FUNCTION_BLOCK "GCS7_M_Motors3W2HL"	// FB 48
TITLE = 3 Motors and 2 HL
//  
//COPYRIGHT:    (C) 1997  BUHLER AG, CH-9240 UZWIL, SWITZERLAND
//
//PRODUCT:      GCS7
//
//TITLE:        FB 48 Machine with 3 Motors and 2 HL 
//
//-------------------------------------------------------------------------
//
//IDENT:        AUTHOR:             DEPT:                       DATE:
//
//FB48.5.0      A. Egli             CT3                         17-Jul-2002
//              New Release with one block 
//              Condition Scraper.InLocal
//FB48.4.0      A. Egli             CT3                         24-Mai-2000
//              Element Scraper (FB11)
//              Mode Separator
//FB48.3.1      A. Egli             CT3                         30-Nov-1999
//              StFault = StCode 32
//FB48.3.0      A. Egli             CT3                         11-Oct-1999
//              Local data reduced 
//FB48.2B       K. Tischer          MU664                       06-Mrz-1999
//              CC FC2 not UC FC2
//FB48.2A       A. Egli             CT3                         04-Mai-1998
//              StFault = StCode 32
//FB48.1A       A.Egli              AEE61                       12-Nov-1997
//              1st Release in S7
//
//-------------------------------------------------------------------------
//
//PURPOSE:      MANUAL : see [LL.M3HxxMAN]
//
//RESTRICTIONS: S7
//              ACCU2: Pointer to dynamic datas of the machine
//              ACCU1: Pointer to parameter datas of the machine
//
//-------------------------------------------------------------------------
//
//
AUTHOR : EA
FAMILY : GCS7LL
NAME : Ma3M2HL
VERSION : 5.0
VAR
  Ma : UDT 20480;
  Motor1 : FB 12;	//Element
  Motor2 : FB 12;	//Element
  Motor3 : FB 12;	//Element
  HLLow : FB 14;	//Element
  HLInlet : FB 14;	//Element
  Scraper : FB 11;	//Element
END_VAR
VAR_TEMP
  tmpFaultStop : BOOL ;
  tmpFaultSum : BOOL ;
  tmpNext : BOOL ;
  tmpLocal : BOOL ;
  tmpEnable : BOOL ;
  tmpSeqStop : BOOL ;
  tmpLenDyn : INT ;
END_VAR
BEGIN
NETWORK
TITLE =
      L     10;
      T     #tmpLenDyn;
NETWORK
TITLE = PC Control
//=== Test Object number =====================
      L     "SYS_DirectCtrlDB".PC.ObjectNo;	//PCControl.ObjectNo
      L     #Ma.Par.ParObjectNo;	//Input ObjectNo
      <>I;
      JC    aEnd;
//=== Test OType      ========================
      L     2048;	//Input object type
      L     "SYS_DirectCtrlDB".PC.ObjectType;	//PCControl.ObjectType
      <>I;
      JC    aEnd;
//=== Test Handshake =========================
      A     "SYS_DirectCtrlDB".PC.Hsk.FExamine;	// Handshake.FExamine
      JC    aExa;
      A     "SYS_DirectCtrlDB".PC.Hsk.FDefineCmd;	// Handshake.FDefineCmd
      O     "SYS_DirectCtrlDB".PC.Hsk.FDefinePara;	// Handshake.FDefinePara
      JC    aCmd;
aIni: L     2;	// FcInit
      UC    "SYS_DirectCtrl";
      JU    aEnd;
// Write new commands from PC to Interface of group 
aCmd: A     "SYS_DirectCtrlDB".PC.Cmd1[0];	//Cmd1[0]=CmdOnM1
      S     #Ma.CmdOn;
      S     #Ma.InDisableM2;
      S     #Ma.InDisableM3;
      A     "SYS_DirectCtrlDB".PC.Cmd1[1];	//Cmd1[1]=CmdOnM2
      R     #Ma.InDisableM2;
      S     #Ma.CmdOn;
      A     "SYS_DirectCtrlDB".PC.Cmd2[1];	//Cmd2[1]=CmdOffM2
      S     #Ma.InDisableM2;
      A     "SYS_DirectCtrlDB".PC.Cmd1[2];	//Cmd1[2]=CmdOnM3
      R     #Ma.InDisableM3;
      S     #Ma.CmdOn;
      A     "SYS_DirectCtrlDB".PC.Cmd2[2];	//Cmd2[2]=CmdOffM3
      S     #Ma.InDisableM3;
      A     "SYS_DirectCtrlDB".PC.Cmd1[8];	//Cmd1[8]=CmdOff
      S     #Ma.CmdOff;
      A     "SYS_DirectCtrlDB".PC.Cmd1[9];	//Cmd1[9]=CmdOn
      S     #Ma.CmdOn;
      R     #Ma.InDisableM2;
      R     #Ma.InDisableM3;
      A     "SYS_DirectCtrlDB".PC.Cmd1[10];	//Cmd1[10]=CmdNext
      S     #Ma.CmdNext;
      A     "SYS_DirectCtrlDB".PC.Cmd1[11];	//Cmd1[11]=CmdFaultReset
      S     #Ma.CmdFaultReset;
      A     "SYS_DirectCtrlDB".PC.Cmd1[13];	//Cmd1[13]=CmdManualOn
      S     #Ma.InManual;
      A     "SYS_DirectCtrlDB".PC.Cmd2[13];	//Cmd1[13]=CmdManualOff
      R     #Ma.InManual;
      AN    "SYS_DirectCtrlDB".PC.Hsk.FDefinePara;	// Handshake.FDefinePara
      JC    aIni;
      JU    aIni;
aExa: TAR2;	// Address Dynamic data
      T     "SYS_DirectCtrlDB".GC.InDynAddr;	// -->PCControl.GC.InDynAddr
      L     #tmpLenDyn;	// Length Dynamic data
      T     "SYS_DirectCtrlDB".GC.InDynLen;	// -->PCControl.GC.InDynLen
      L     0;
      T     "SYS_DirectCtrlDB".GC.InParaAddr;	// -->PCControl.GC.InParaAddr
      T     "SYS_DirectCtrlDB".GC.InParaLen;	// -->PCControl.GC.InParaLen
      L     1;	// Code FcExamine
      UC    "SYS_DirectCtrl";
      L     10;	//Revision
      T     "SYS_DirectCtrlDB".GC.Revision;
aEnd: NOP   0;
NETWORK
TITLE = Interlocking
//===Global Group Orders===
      A     "GCS7_Gr_OutManualOn";	//Gr.OutManualOn
      S     #Ma.InManual;
      A     "GCS7_Gr_OutManualOff";	//Gr.OutManualOff
      R     #Ma.InManual;
      A     #Ma.InManual;
      S     "GCS7_Gr_InManual";	//Gr.InManual
      A     #Ma.CmdNext;
      AN    #Ma.InManual;
      O     #Ma.CmdOn;
      =     #tmpNext;
      A     #Ma.InManual;
      ON    #Ma.InLocal;
      A     #Ma.InEnable;
      AN    #Ma.CmdOff;
      =     #tmpEnable;
      A     #Ma.InSeqStop;
      AN    #Ma.InManual;
      =     #tmpSeqStop;
//--- Fault----
      A     #Motor1.StFault;
      O     #Motor2.StFault;
      O     #Motor3.StFault;
      O     #HLLow.StFault;
      O     #HLInlet.StFault;
      O     #Scraper.StFault;
      =     #tmpFaultSum;
//--- Next
      A(;
      A     #Motor2.StStartedFwd;
      ON    #Ma.Par.ParTypeSeparator;
      );
      A     #tmpNext;
      S     #Motor1.CmdNext;
      A     #Motor1.StStartedFwd;
      O     #Ma.Par.ParTypeSeparator;
      A     #tmpNext;
      S     #Motor2.CmdNext;
      S     #Motor3.CmdNext;
      A     #tmpNext;
      S     #Scraper.CmdNext;
//--- Interlocking Motors
//Motor1
      A     #tmpEnable;
      O     #Ma.Par.ParMotor1IsFan;
      =     #Motor1.InEnableFwd;
// 
      A     #tmpSeqStop;
      ON    #tmpEnable;
      A     #Motor2.StStopped;
      O;
      AN    #Ma.Par.ParMotor1IsFan;
      A     #tmpSeqStop;
      =     #Motor1.InSeqStop;
//Motor2
      AN    #HLLow.StFault;
      ON    #Ma.Par.ParWithHLLow;
      A(;
      A     #Motor1.StStartedFwd;
      O     #Ma.Par.ParTypeSeparator;
      );
      AN    #Ma.InDisableM2;
      A     #tmpEnable;
      =     #Motor2.InEnableFwd;
      A     #tmpSeqStop;
      =     #Motor2.InSeqStop;
//Motor3 
      A     #Motor2.InEnableFwd;
      A     #Motor2.StStartedFwd;
      O     #Ma.Par.ParTypeSeparator;
      A     #Motor1.StStartedFwd;
      AN    #Ma.InDisableM3;
      A     #tmpEnable;
      =     #Motor3.InEnableFwd;
      A     #tmpSeqStop;
      =     #Motor3.InSeqStop;
//Scraper
      A     #Motor2.StStartedFwd;
      A     #tmpEnable;
      =     #Scraper.InEnable;
      A     #tmpSeqStop;
      =     #Scraper.InSeqStop;
// 
//--- Local mode --
      A     #Ma.InLocal;
      AN    #Ma.InManual;
      =     #Motor1.InLocal;
      =     #Motor2.InLocal;
      =     #Motor3.InLocal;
      =     #HLLow.InLocal;
      =     #HLInlet.InLocal;
      =     #Scraper.InLocal;
//--- Fault Reset -------------
      A     #Ma.CmdFaultReset;
      S     #Motor1.CmdFaultReset;
      S     #Motor2.CmdFaultReset;
      S     #Motor3.CmdFaultReset;
      S     #HLLow.CmdFaultReset;
      S     #HLInlet.CmdFaultReset;
      S     #Scraper.CmdFaultReset;
// 
//--- Monitoring Level
      SET;
      S     #HLLow.InMonFalse;
      S     #HLInlet.InMonFalse;
NETWORK
TITLE = Call Motor1
      CALL  #Motor1;
NETWORK
TITLE = Call Motor2
      CALL  #Motor2;
NETWORK
TITLE = Call Motor3
      AN    #Ma.Par.ParWithMotor3;
      JC    el4;
      CALL  #Motor3;
NETWORK
TITLE = Call Digital Input: HLLow
el4:  AN    #Ma.Par.ParWithHLLow;
      JC    el5;
      CALL  #HLLow;
NETWORK
TITLE = Call Digital Input: HLInlet
el5:  AN    #Ma.Par.ParWithHLInlet;
      JC    el6;
      CALL  #HLInlet;
NETWORK
TITLE = Call Digital Output: Scraper
el6:  AN    #Ma.Par.ParWithScraper;
      JC    SPen;
      CALL  #Scraper;
SPen: NOP   0;
NETWORK
TITLE = Actual State
// StFault
      A     #tmpFaultSum;
      =     #Ma.StFault;
// StStopped
      A     #Motor3.StStopped;
      ON    #Ma.Par.ParWithMotor3;
      A     #Motor1.StStopped;
      A     #Motor2.StStopped;
      AN    #Ma.StFault;
      =     #Ma.StStopped;
// StStarted
      A     #Motor3.StStartedFwd;
      ON    #Ma.Par.ParWithMotor3;
      A     #Motor1.StStartedFwd;
      A     #Motor2.StStartedFwd;
      AN    #Ma.StFault;
      =     #Ma.StStarted;
// StStopping
      A     #Motor1.InSeqStop;
      O     #Motor2.InSeqStop;
      O     #Motor3.InSeqStop;
      AN    #Ma.StStarted;
      AN    #Ma.StStopped;
      AN    #Ma.StFault;
      =     #Ma.StStopping;
// StStarting
      AN    #Ma.StStopped;
      AN    #Ma.StStarted;
      AN    #Ma.StStopping;
      AN    #Ma.StFault;
      =     #Ma.StStarting;
NETWORK
TITLE = State Code
// State             StCode
// -------------------------
// StFault             32
// StStopped            1
// StStarting           2
// StStarted.Wait       3
// StStarted.Feeding    4
// StEmptying           5
// StEmptied            6
// StStopping           7
      A     #Ma.StStopped;
      L     1;	//Code=StStopped
      JC    Code;
      A     #Ma.StStarted;
      L     3;	//Code=StStarted
      JC    Code;
      A     #Ma.StStarting;
      L     2;	//Code=StStarting
      JC    Code;
      A     #Ma.StStopping;
      L     7;	//Code=StStopping 
      JC    Code;
      L     32;	//3.1: Code=StFault 
Code: L     #Ma.StCode;	// Old state code
      TAK;
      T     #Ma.StCode;	// Save state code
      <>I;
      L     3;
      CC    "SYS_CBitCtrl";	//Set change bit
NETWORK
TITLE = Global End
      CLR;	//---Clear all commands
      =     #Ma.CmdOn;
      =     #Ma.CmdOff;
      =     #Ma.CmdNext;
      =     #Ma.CmdFaultReset;
END_FUNCTION_BLOCK

FUNCTION_BLOCK "GCS7_M_MDDX"	// FB 49
TITLE = MDDx Newtronic Roll Stand
//  
//COPYRIGHT:    (C) 1999  BUHLER AG, CH-9240 UZWIL, SWITZERLAND
//
//PRODUCT:      GCS7
//
//TITLE:        FB 49 Machine MDDx Newtronic Roll Stand
//              (GCPROVB Revision 11)
//-------------------------------------------------------------------------
//
//IDENT:        AUTHOR:             DEPT:                       DATE:
//
//FB49.5.3      A. Egli             CT3                         15-Aug-2007
//              MDDX.OutComFault stops motors
//FB49.5.2      A. Egli             CT3                         15-Feb-2007
//              Stop Motors when alarm 14 or 15
//FB49.5.1      Ph. Enger           MU664                       21-Sep-2004
//              Interlocking with BackupHL corrected
//FB49.5.0      Ph. Enger           MU664                       16-Sep-2004
//              New configuration ParB1
//FB49.4.0      A. Egli             CT3                         28-Jul-2004
//              New Version of FB35
//FB49.3.1      A. Egli             CT3                         05-Mai-2004
//              CmdOff in manual mode
//FB49.3.0      A. Egli             CT3                         17-Jul-2002
//              New Release with one block 
//FB49.2.2      A. Egli             CT3                         18-Mai-2000
//              CBIT: UC changed with CC 
//FB49.2.1      S. Kalberer         CT3                         29-Nov-1999
//              HLInlet: InOverwriteHL function to InMonFalse not InLocal
//FB49.2.0      A. Egli             CT3                         11-Oct-1999
//              Local data reduced 
//FB49.1A       S. Kalberer         CT3                         30-Jul-1999
//              1st Release in S7
//
//-------------------------------------------------------------------------
//
//PURPOSE:      MANUAL : see [LL.ROXENMAN]
//
//RESTRICTIONS: S7
//              ACCU2: Pointer to dynamic datas of the machine
//              ACCU1: Pointer to parameter datas of the machine
//
//-------------------------------------------------------------------------
//
//
AUTHOR : EA
FAMILY : GCS7LL
NAME : MDDxNtro
VERSION : 5.3
VAR
  Ma : UDT 20490;
  RollsUp : FB 12;	//Element
  RollsLow : FB 12;	//Element
  HLInlet : FB 14;	//Element
  HLBackUp : FB 14;	//Element
  HLOutlet : FB 14;	//Element
  CollectAlarm : FB 14;	//Element
  MddLC : FB 35;	//Element
  FU_Feedroll : FB 14;	//Element FU Feedroll [3.0]
END_VAR
VAR_TEMP
  tmpFaultSum : BOOL ;
  tmpWarning : BOOL ;
  tmpStarted : BOOL ;
  tmpNext : BOOL ;
  tmpLocal : BOOL ;
  tmpEnable : BOOL ;
  tmpSeqStop : BOOL ;
  tmpLenDyn : INT ;
END_VAR
BEGIN
NETWORK
TITLE =
      L     10;
      T     #tmpLenDyn;
NETWORK
TITLE = PC Control
//=== Test Object number =====================
      L     "SYS_DirectCtrlDB".PC.ObjectNo;	//PCControl.ObjectNo
      L     #Ma.Par.ParObjectNo;	//Input ObjectNo
      <>I;
      JC    aEnd;
//=== Test OType      ========================
      L     2049;	//Input object type
      L     "SYS_DirectCtrlDB".PC.ObjectType;	//PCControl.ObjectType
      <>I;
      JC    aEnd;
//=== Test Handshake =========================
      A     "SYS_DirectCtrlDB".PC.Hsk.FExamine;	// Handshake.FExamine
      JC    aExa;
      A     "SYS_DirectCtrlDB".PC.Hsk.FDefineCmd;	// Handshake.FDefineCmd
      O     "SYS_DirectCtrlDB".PC.Hsk.FDefinePara;	// Handshake.FDefinePara
      JC    aCmd;
aIni: L     2;	// FcInit
      UC    "SYS_DirectCtrl";
      JU    aEnd;
// Write new commands from PC to Interface of group 
aCmd: A     "SYS_DirectCtrlDB".PC.Cmd1[1];	//Cmd1[1]=CmdEnableEngageOn
      S     #Ma.InEnableEngage;
      A     "SYS_DirectCtrlDB".PC.Cmd2[1];	//Cmd2[1]=CmdEnableEngageOff
      R     #Ma.InEnableEngage;
      A     "SYS_DirectCtrlDB".PC.Cmd1[2];	//Cmd1[2]=CmdResDischargeOn
      S     #Ma.InRestdischarge;
      A     "SYS_DirectCtrlDB".PC.Cmd2[2];	//Cmd2[2]=CmdRestDischargeOff
      R     #Ma.InRestdischarge;
      A     "SYS_DirectCtrlDB".PC.Cmd1[3];	//Cmd1[3]=CmdOverwriteHLOn
      S     #Ma.InOverrideHL;
      A     "SYS_DirectCtrlDB".PC.Cmd2[3];	//Cmd2[3]=CmdOverwriteHLOff
      R     #Ma.InOverrideHL;
      A     "SYS_DirectCtrlDB".PC.Cmd1[8];	//Cmd1[8]=CmdOff
      S     #Ma.CmdOff;
      A     "SYS_DirectCtrlDB".PC.Cmd1[9];	//Cmd1[9]=CmdOn
      S     #Ma.CmdOn;
      A     "SYS_DirectCtrlDB".PC.Cmd1[10];	//Cmd1[10]=CmdNext
      S     #Ma.CmdNext;
      A     "SYS_DirectCtrlDB".PC.Cmd1[11];	//Cmd1[11]=CmdFaultReset
      S     #Ma.CmdFaultReset;
      A     "SYS_DirectCtrlDB".PC.Cmd1[13];	//Cmd1[13]=CmdManualOn
      S     #Ma.InManual;
      A     "SYS_DirectCtrlDB".PC.Cmd2[13];	//Cmd1[13]=CmdManualOff
      R     #Ma.InManual;
      AN    "SYS_DirectCtrlDB".PC.Hsk.FDefinePara;	// Handshake.FDefinePara
      JC    aIni;
      JU    aIni;
aExa: TAR2;	// Address Dynamic data
      T     "SYS_DirectCtrlDB".GC.InDynAddr;	// -->PCControl.GC.InDynAddr
      L     #tmpLenDyn;	// Length Dynamic data
      T     "SYS_DirectCtrlDB".GC.InDynLen;	// -->PCControl.GC.InDynLen
      L     0;
      T     "SYS_DirectCtrlDB".GC.InParaAddr;	// -->PCControl.GC.InParaAddr
      T     "SYS_DirectCtrlDB".GC.InParaLen;	// -->PCControl.GC.InParaLen
      L     1;	// Code FcExamine
      UC    "SYS_DirectCtrl";
      L     12;	//Revision
      T     "SYS_DirectCtrlDB".GC.Revision;
aEnd: NOP   0;
NETWORK
TITLE = Interlocking
//===Global Group Orders===
      A     "GCS7_Gr_OutManualOn";	//Gr.OutManualOn
      S     #Ma.InManual;
      A     "GCS7_Gr_OutManualOff";	//Gr.OutManualOff
      R     #Ma.InManual;
      A     #Ma.InManual;
      S     "GCS7_Gr_InManual";	//Gr.InManual
//--- temporary Next ---
      AN    #Ma.StStarting;
      ON    #Ma.InManual;
      O     #Ma.CmdOff;	//[3.1]
      R     #Ma.OutStartMan;
      O     #Ma.CmdOn;
      S     #Ma.OutStartMan;
      A     #Ma.CmdNext;
      AN    #Ma.InManual;
      O     #Ma.OutStartMan;
      =     #tmpNext;
//--- temporary Enable ---
      A(;
      A     #Ma.InEnable;
      AN    #Ma.InLocal;
      AN    #Ma.InManual;
      O;
      A     #Ma.InEnable;
      A     #Ma.InManual;
      AN    #Ma.Par.ParManual;
      O;
      A     #Ma.Par.ParManual;
      A     #Ma.InManual;
      );
      AN    #Ma.CmdOff;
      AN    #MddLC.Par.OutLCAlarm.GrindRollsStandstill;	//[5.2]
      AN    #MddLC.Par.OutLCAlarm.GrindRollsLowStandstill;	//[5.2]
      AN    #MddLC.OutComFault;	//[5.3]
      =     #tmpEnable;
//--- temporary SeqStop ---
      A     #Ma.InSeqStop;
      AN    #Ma.InManual;
      =     #tmpSeqStop;
//--- Fault----
      A     #RollsUp.StFault;
      O     #RollsLow.StFault;
      =     #tmpWarning;
      A     #tmpWarning;
      AN    #Ma.Par.ParWarning;
      O     #HLBackUp.StFault;
      O     #HLInlet.StFault;
      O     #HLOutlet.StFault;
      O     #CollectAlarm.StFault;
      O     #MddLC.StFault;
      O     #FU_Feedroll.StFault;	//[3.0]
      =     #tmpFaultSum;
//--- Next
      A     #HLBackUp.StFalse;	//[5.0]
      ON    #Ma.Par.ParWithHLBackUp;	//[5.1]
      A     #tmpNext;
      S     #RollsLow.CmdNext;
      S     #RollsUp.CmdNext;
//--- Interlocking Motors
//RollsLow
      A     #tmpEnable;
      AN    #tmpSeqStop;	//[5.0]
      =     #RollsLow.InEnableFwd;
// 
      A     #HLBackUp.StFault;	//[5.0]
      A     #HLBackUp.InpTrue;	//[5.0]
      =     #RollsLow.InSeqStop;
//RollsUp
      A     #RollsLow.StStartedFwd;
      ON    #Ma.Par.ParWithRollsLow;
      A     #tmpEnable;
      AN    #tmpSeqStop;	//[5.0]
      =     #RollsUp.InEnableFwd;
      A     #HLBackUp.StFault;	//[5.0]
      A     #HLBackUp.InpTrue;	//[5.0]
      =     #RollsUp.InSeqStop;
//--- Local mode --
      A     #Ma.InLocal;
      AN    #Ma.InManual;
      =     #RollsLow.InLocal;
      =     #RollsUp.InLocal;
      =     #HLBackUp.InLocal;
      =     #HLOutlet.InLocal;
      =     #CollectAlarm.InLocal;
      =     #MddLC.InLocal;
      =     #FU_Feedroll.InLocal;	//[3.0]
//        U     #Ma.InLocal;      // 2.1
//        UN    #Ma.InManual;     // 2.1
//        O     #Ma.InOverwriteHL; // 2.1 
      =     #HLInlet.InLocal;
//--- Fault Reset -------------
      A     #Ma.CmdFaultReset;
      S     #RollsLow.CmdFaultReset;
      S     #RollsUp.CmdFaultReset;
      S     #HLInlet.CmdFaultReset;
      S     #HLBackUp.CmdFaultReset;
      S     #HLOutlet.CmdFaultReset;
      S     #CollectAlarm.CmdFaultReset;
      S     #MddLC.CmdFaultReset;
      S     #FU_Feedroll.CmdFaultReset;	//[3.0]
//--- Monitoring 
      AN    #Ma.InOverrideHL;	// 2.1
      O     #Ma.Par.ParB1;	//[5.0]
      =     #HLInlet.InMonFalse;	// 2.1
      AN    #Ma.Par.ParB1;	//[5.0]
      AN    #Ma.InOverrideHL;	//[5.0]
      =     #HLInlet.InPreAlarmFalse;	//[5.0]
// 
      A     #HLInlet.OutFlagPos;	//[5.0] 
      AN    #HLInlet.OutTimeoutTime;	//[5.0] 
      A     #Ma.Par.ParB1;	//[5.0]
      S     #HLInlet.CmdRunTimeoutTime;	//[5.0]
// 
      SET;
      S     #HLBackUp.InMonFalse;
      S     #HLOutlet.InMonFalse;
      S     #CollectAlarm.InMonTrue;
//Startup done
      A     #RollsUp.StStartedFwd;
      O     #RollsUp.StFault;
      A(;
      A     #RollsLow.StStartedFwd;
      O     #RollsLow.StFault;
      ON    #Ma.Par.ParWithRollsLow;
      );
      =     #Ma.OutStartupDone;
      A     #RollsLow.StStartedFwd;
      ON    #Ma.Par.ParWithRollsLow;
      A     #RollsUp.StStartedFwd;
      =     #tmpStarted;
//--- Serial Communication Handling
// EnableEngage
      A     #Ma.InEnable;
      AN    #Ma.InLocal;
      AN    #Ma.InManual;
      O     #Ma.InEnableEngage;
      =     #MddLC.InEnableEngage;
//  RestDischarge
      A     #Ma.InRestdischarge;
      =     #MddLC.InRestdischarge;
NETWORK
TITLE = Call RollsUp
      CALL  #RollsUp;
NETWORK
TITLE = Call RollsLow
      AN    #Ma.Par.ParWithRollsLow;
      JC    el3;
      CALL  #RollsLow;
NETWORK
TITLE = Call Digital Input: HLInlet
el3:  AN    #Ma.Par.ParWithHLInlet;
      JC    el4;
      CALL  #HLInlet;
NETWORK
TITLE = Call Digital Input: HLBackUp
el4:  AN    #Ma.Par.ParWithHLBackUp;
      JC    el5;
      CALL  #HLBackUp;
NETWORK
TITLE = Call Digital Input: HLOutlet
el5:  AN    #Ma.Par.ParWithHLOutlet;
      JC    el6;
      CALL  #HLOutlet;
NETWORK
TITLE = Call Digital Input: CollectAlarm
el6:  AN    #Ma.Par.ParWithCollectAlarm;
      JC    el7;
      CALL  #CollectAlarm;
NETWORK
TITLE = Call MDDx Serial Communication: MddLC
el7:  AN    #Ma.Par.ParWithMddLC;
      JC    el8;
      CALL  #MddLC;
NETWORK
TITLE = Call MDDx Serial Communication: MddLC
el8:  AN    #Ma.Par.ParWithFU_FeedRoll;	//[3.0]
      JC    StJ0;
      CALL  #FU_Feedroll;
NETWORK
TITLE = Actual State
// StFault
StJ0: A     #tmpFaultSum;
      =     #Ma.StFault;
// StWarning
      A     #tmpWarning;
      A     #Ma.Par.ParWarning;
      AN    #Ma.StFault;
      O     #MddLC.StWarning;
      =     #Ma.StWarning;
// StStopped
      A     #RollsLow.StStopped;
      ON    #Ma.Par.ParWithRollsLow;
      A     #RollsUp.StStopped;
      AN    #Ma.StFault;
      =     #Ma.StStopped;
// StStarted
      A     #tmpStarted;
      AN    #Ma.StFault;
      AN    #Ma.StStopped;
      =     #Ma.StStarted;
// StStopping
      A     #RollsUp.InSeqStop;
      O     #RollsLow.InSeqStop;
      AN    #Ma.StStarted;
      AN    #Ma.StStopped;
      AN    #Ma.StFault;
      AN    #Ma.StWarning;
      =     #Ma.StStopping;
// StStarting
      AN    #Ma.StStopped;
      AN    #Ma.StStarted;
      AN    #Ma.StStopping;
      AN    #Ma.StFault;
      AN    #Ma.StWarning;
      =     #Ma.StStarting;
NETWORK
TITLE = State Code
// State     StCode
// ----------------------
// StFault32
// StStopped    1
// StStarting   2
// StStarted   3
// StStopping  7
// StWarning8
      A     #Ma.StStopped;
      L     1;	//Code=StStopped
      JC    Code;
      A     #Ma.StStarted;
      L     3;	//Code=StStarted
      JC    Code;
      A     #Ma.StWarning;
      L     8;	//Code=StWarning 
      JC    Code;
      A     #Ma.StStarting;
      L     2;	//Code=StStarting
      JC    Code;
      A     #Ma.StStopping;
      L     7;	//Code=StStopping 
      JC    Code;
      L     32;	//Code=StFault 
Code: L     #Ma.StCode;	// Old state code
      TAK;
      T     #Ma.StCode;	// Save state code
      <>I;
      L     3;
      CC    "SYS_CBitCtrl";	//Set change bit [REL 2.2]
NETWORK
TITLE = Global End
      CLR;	//---Clear all commands
      =     #Ma.CmdOn;
      =     #Ma.CmdOff;
      =     #Ma.CmdNext;
      =     #Ma.CmdFaultReset;
END_FUNCTION_BLOCK

FUNCTION_BLOCK "GCS7_M_Motor6Mon"	// FB 50
TITLE = Motor with 6 digital input
//  
//COPYRIGHT:    (C) 1997  BUHLER AG, CH-9240 UZWIL,  SWITZERLAND
//
//PRODUCT:      GCS7
//
//TITLE:        FB 50 MACHINE-CONTROL:Motor with 6 Digital input 
//              GCPROVB Revision >=12
// 
//-------------------------------------------------------------------------
//
//IDENT:        AUTHOR:             DEPT:                       DATE:
//FB50.8.6      A.Egli              BASE                        10-Apr-2008
//              - Init if download DB
//              - Condition MonX.InLocal 
//FB50.8.5      Ph. Engler          GP92                        23-Aug-2007
//              Machine status: StStarting how long the monitoring elements
//FB50.8.5      Ph. Engler          GP92                        23-Aug-2007
//              Machine status: StStarting how long the monitoring elements
//                              aren't in the correct status
//FB50.8.4      A.Egli              CT3                         20-Feb-2006
//              EBM-Test procedure: - Include als the EBMInput to the test
//                                  - Manual and local mode also integrated 
//              (Tested Ph.Engler, GP92,24-Aug-2005 )
//FB50.8.3      A.Egli              CT3                         09-Mar-2005
//              Send CmdFaultReset only with positve edge to elements  
//FB50.8.2      A.Egli              CT3                         20-Sep-2004 
//              Delay time before and between 2 single tests of EBM  
//FB50.8.1      A.Egli              CT3                         20-Jul-2004
//              tmpLenDyn is 12 and not 10
//FB50.8.0      A.Egli              CT3                         25-Mai-2004
//              ParMon4IsSM
//FB50.7.6      A.Egli              CT3                         15-Apr-2004
//              Test with Hardware 
//FB50.7.5      A.Egli              CT3                         18-Mar-2004
//              InpControlEBM 
//FB50.7.4      K. Tischer          CT3                         13-Feb-2004
//              interlocking without Mon1 
//FB50.7.3      K. Tischer          CT3                         30-Jan-2004
//              Correct monitoring Mon4 
//FB50.7.2      K. Tischer          CT3                         14-Jan-2004
//              Revision=11 
//FB50.7.1      K. Tischer          CT3                         02-Dec-2003
//              new 6 DI and supported EBM3003 
//FB50.7.0      K. Tischer          CT3                         01-Dec-2003
//              new 6 DI and supported EBM3003 
//FB50.6.2      A. Egli             CT3                         22-Sep-2003
//              Interlocking Mon4.StFalse when Mon4 is HL
//FB50.6.1      A. Egli             CT3                         16-Mai-2003
//              Interlocking if Mon1 is HL
//              Send CmdOff to Motor
//FB50.6.0      A. Egli             CT3                         17-Jun-2002
//              New Release with one block 
//              Interlocking if Mon1 is HL
//FB50.5.0      A. Egli             CT3                          1-Feb-2002
//              -HLInlet renamed as Mon4
//              -ParMon4StopByFault,ParMon4IsLS
//FB50.4.0      A. Egli             CT3                         15-Jan-2002
//              HLIntet as Warning Element
//FB50.3.1      A. Egli             CT3                         23-Oct-2001
//              Manual Mode: no interlocking with InSeqStop
//FB50.3.0      A. Egli             CT3                         11-Oct-1999
//              Local data reduced 
//FB50.2C       A. Egli             CT3                         03-Juni-1999
//              Manual Mode
//FB50.2B       K. Tischer          MU664                       06-Mrz-1999
//              CC FC2 not UC FC2
//FB50.2A       A. Egli             CT3                         04-Mai-1998
//              StFault = StCode 32
//FB50.1A       A.Egli              AEE61                       5-Jul-1997
//              1st Release in S7
//
//-------------------------------------------------------------------------
//
//PURPOSE:      MANUAL : see [LL.M4IxxMAN]
//
//RESTRICTIONS: S7
//
//              GCPROVB Revision >=5
//-------------------------------------------------------------------------
//
AUTHOR : EA
FAMILY : GCS7LL
NAME : M_6DI
VERSION : 8.6
VAR
  Ma : UDT 20500;
  Mon1 : FB 14;	//Element Mon 1 optional
  Mon2 : FB 14;	//Element Mon 2
  Mon3 : FB 14;	//Element Mon 3 optional
  Mon4 : FB 14;	//Element Mon 4 optional
  Mon5 : FB 14;	//Element Mon 5 optional [7.0]
  Mon6 : FB 14;	//Element Mon 6 optional [7.0]
  Motor : FB 12;	//Element Motor
END_VAR
VAR_TEMP
  tmpFaultStop : BOOL ;
  tmpFaultSum : BOOL ;
  tmpEnable : BOOL ;
  tmpLocal : BOOL ;
  tmpLenDyn : INT ;
  tmpOK : BOOL ;
  tmpTestTime : INT ;
  tmpMonElOk : BOOL ;
END_VAR
BEGIN
NETWORK
TITLE =
      L     12;
      T     #tmpLenDyn;	//[8.1]
NETWORK
TITLE = PC Control
//=== Test Object number =====================
      L     "SYS_DirectCtrlDB".PC.ObjectNo;	//PCControl.ObjectNo
      L     #Ma.Par.ParObjectNo;	//Input ObjectNo
      <>I;
      JC    aEnd;
//=== Test OType      ========================
      L     2050;	//Input object type
      L     "SYS_DirectCtrlDB".PC.ObjectType;	//PCControl.ObjectType
      <>I;
      JC    aEnd;
//=== Test Handshake =========================
      A     "SYS_DirectCtrlDB".PC.Hsk.FExamine;	// Handshake.FExamine
      JC    aExa;
      A     "SYS_DirectCtrlDB".PC.Hsk.FDefineCmd;	// Handshake.FDefineCmd
      O     "SYS_DirectCtrlDB".PC.Hsk.FDefinePara;	// Handshake.FDefinePara
      JC    aCmd;
aIni: L     2;	// FcInit
      UC    "SYS_DirectCtrl";
      JU    aEnd;
// Write new commands from PC to Interface of group 
aCmd: A     "SYS_DirectCtrlDB".PC.Cmd1[8];	//Cmd1[8]=CmdOff
      S     #Ma.CmdOff;
      A     "SYS_DirectCtrlDB".PC.Cmd1[9];	//Cmd1[9]=CmdOn
      S     #Ma.CmdOn;
      A     "SYS_DirectCtrlDB".PC.Cmd1[10];	//Cmd1[10]=CmdNext
      S     #Ma.CmdNext;
      A     "SYS_DirectCtrlDB".PC.Cmd1[11];	//Cmd1[11]=CmdFaultReset
      S     #Ma.CmdFaultReset;
      A     "SYS_DirectCtrlDB".PC.Cmd1[13];	//Cmd1[13]=CmdManualOn
      S     #Ma.InManual;
      A     "SYS_DirectCtrlDB".PC.Cmd1[6];	//Cmd1[6]=CmdManSlowOn
      S     #Motor.InOutManSlow;
      A     "SYS_DirectCtrlDB".PC.Cmd1[7];	//Cmd1[7]=CmdManRevOn
      S     #Motor.InOutManRev;
      A     "SYS_DirectCtrlDB".PC.Cmd2[13];	//Cmd2[13]=CmdManualOff
      R     #Ma.InManual;
      A     "SYS_DirectCtrlDB".PC.Cmd2[6];	//Cmd2[6]=CmdManSlowOff
      R     #Motor.InOutManSlow;
      A     "SYS_DirectCtrlDB".PC.Cmd2[7];	//Cmd2[7]=CmdManRevOff
      R     #Motor.InOutManRev;
      JU    aIni;
aExa: TAR2;	// Address Dynamic datas
      T     "SYS_DirectCtrlDB".GC.InDynAddr;	// -->PCControl.GC.InDynAddr
      L     #tmpLenDyn;	// Length Dynamic data
      T     "SYS_DirectCtrlDB".GC.InDynLen;	// -->PCControl.GC.InDynLen
      L     0;
      T     "SYS_DirectCtrlDB".GC.InParaAddr;	// -->PCControl.GC.InParaAddr
      T     "SYS_DirectCtrlDB".GC.InParaLen;	// -->PCControl.GC.InParaLen
      L     1;	// Code FcExamine
      UC    "SYS_DirectCtrl";
      L     12;	//Revision
      T     "SYS_DirectCtrlDB".GC.Revision;
aEnd: NOP   0;
NETWORK
TITLE = function test [7.0]
      L     720;	//[8.2] 
      T     #tmpTestTime;	//[8.2] 
      AN    #Ma.Par.ParEBM;
      JC    FCT0;
      A     #Ma.InLocal;
      AN    #Ma.InManual;
      =     #tmpLocal;
      L     0;
      L     #Ma.OutTestTime;
      >=I;
      O     #Ma.CmdTestEBM;
      R     #Ma.InfBMTopOk;
      R     #Ma.InfBMBottomOk;
      R     #Ma.InfSMOk;
      R     #Ma.CmdTestEBM;
      L     #tmpTestTime;	//s = 12min 
      JC    FCT;
      AN    #Motor.StStartedFwd;	//[8.2] 
      AN    #Motor.StStartedRev;	//[8.2] 
      AN    #Ma.InfSMOk;	//[8.2] 
      L     #tmpTestTime;	//[8.2] 
      JC    FCT;	//[8.2] 
      L     #Ma.OutTestTime;
      AN    "GCS7_Gr_OutTick1s";	// Gr.OutTick1s
      JC    FCT;
      +     -1;
FCT:  T     #Ma.OutTestTime;
// function test SM
      L     #tmpTestTime;	//[8.2] 
      L     #Ma.OutTestTime;	//[8.2] 
      -I;	//[8.2] 
      L     35;	//[8.2] 
      >=I;	//[8.2] 
      A     #Ma.InpControlEBM;	//[7.5]
      AN    #Ma.OutpFaultReset;	//[7.5]
      AN    #Ma.StFault;	//[7.5]
      O     #Ma.OutpFcttst_SM;	//[7.5]
      AN    #Ma.InfSMOk;
      AN    #Mon1.InLocal;
      AN    #Ma.StStopped;	//[8.2]
      =     #Ma.OutpFcttst_SM;
// function test ok SM
      A     #Ma.OutpFcttst_SM;
      A(;
      ON    #Mon6.InpTrue;
      ON    #Ma.Par.ParWithMon6;
      );
      AN    #Ma.InpControlEBM;	//[7.5]
      =     #tmpOK;	//[7.5]
      A     #tmpOK;	//[7.5]
      AN    #Ma.InfSMOk;	//[7.5]
      S     #Ma.InfSMOk;
      S     #Ma.OutFaultResetFcttst;	//[7.5]
      JCN   BTJ1;	//[8.2] 
      L     #tmpTestTime;	//[8.2] s = 12min 
      T     #Ma.OutTestTime;	//[8.2] 
BTJ1: NOP   0;	//[8.2] 
// function test BM top
      L     #tmpTestTime;	//[8.2] s = 12min 
      L     #Ma.OutTestTime;	//[8.2] 
      -I;	//[8.2] 
      L     5;	//[8.2] 
      >=I;	//[8.2] 
      AN    #Ma.OutpFaultReset;	//[7.5]
      A     #Ma.InpControlEBM;	//[7.5]
      AN    #Ma.StFault;	//[7.5]
      O     #Ma.OutpFcttst_BM_Top;	//[7.5]
      AN    #Ma.InfBMTopOk;
      A     #Ma.InfSMOk;	//[7.6]
      AN    #Mon1.InLocal;
      =     #Ma.OutpFcttst_BM_Top;
// function test ok
      A     #Ma.OutpFcttst_BM_Top;
      AN    #Mon2.InpTrue;
      AN    #Ma.InpControlEBM;	//[7.5]
      =     #tmpOK;	//[7.5]
      A     #tmpOK;	//[7.5]
      AN    #Ma.InfBMTopOk;	//[7.5]
      S     #Ma.InfBMTopOk;
      S     #Ma.OutFaultResetFcttst;	//[7.5]
      JCN   BTJ2;	//[8.2] 
      L     #tmpTestTime;	//[8.2] s = 12min 
      T     #Ma.OutTestTime;	//[8.2] 
BTJ2: NOP   0;	//[8.2] 
// function test BM Bottom
      L     #tmpTestTime;	//[8.2] s = 12min 
      L     #Ma.OutTestTime;	//[8.2] 
      -I;	//[8.2] 
      L     5;	//[8.2] 
      >=I;	//[8.2] 
      A     #Ma.InpControlEBM;	//[7.5]
      AN    #Ma.OutpFaultReset;	//[7.5]
      AN    #Ma.StFault;	//[7.5]
      O     #Ma.OutpFcttst_BM_Bottom;	//[7.5]
      AN    #Ma.InfBMBottomOk;
      A     #Ma.InfBMTopOk;
      A     #Ma.InfSMOk;	//[7.6]
      AN    #Mon1.InLocal;
      =     #Ma.OutpFcttst_BM_Bottom;
// function test ok BM Bottom 
      A     #Ma.OutpFcttst_BM_Bottom;
      A(;
      ON    #Mon4.InpTrue;
      ON    #Ma.Par.ParWithMon4;
      );
      AN    #Ma.InpControlEBM;	//[7.5]
      =     #tmpOK;	//[7.5]
      A     #tmpOK;	//[7.5]
      AN    #Ma.InfBMBottomOk;	//[7.5]
      S     #Ma.InfBMBottomOk;
      S     #Ma.OutFaultResetFcttst;	//[7.5]
FCT0: NOP   0;
NETWORK
TITLE = Interlocking
//===Global Group Orders===
      A     "GCS7_Gr_OutManualOn";	//Gr.OutManualOn
      S     #Ma.InManual;
      A     "GCS7_Gr_OutManualOff";	//Gr.OutManualOff
      R     #Ma.InManual;
      A     #Ma.InManual;
      S     "GCS7_Gr_InManual";	//Gr.InManual
// 
      A     "GCS7_Gr_OutFaultReset";	// OutFaultReset
      S     #Ma.CmdFaultReset;
//--- Fault----
      A     #Ma.Par.ParMon1StopByFault;
      A     #Mon1.StFault;
      O     #Mon2.StFault;
      O     #Mon3.StFault;
      O(;	//[5.0]
      A     #Ma.Par.ParMon4StopByFault;	//[5.0]
      O     #Ma.Par.ParMon4IsSM;	//[8.0]
      O     #Ma.Par.ParEBM;	//[7.6]
      A     #Mon4.StFault;	//[5.0]
      );	//[5.0]
      O     #Mon5.StFault;	//[7.0]
      O     #Mon6.StFault;	//[7.0]
      =     #tmpFaultStop;
      A     #Mon4.StFault;	//[4.0]
      AN    #Ma.Par.ParMon4AsWarning;	//[4.0]
      O     #Mon1.StFault;
      O     #Motor.StFault;
      O     #tmpFaultStop;
      =     #tmpFaultSum;
      A     #Mon4.StFault;	//[4.0]
      A     #Ma.Par.ParMon4AsWarning;	//[4.0]
      =     #Ma.OutWarning;	//[4.0]
//--- Motor----
      A     #tmpFaultStop;	//[8.4]
      A     #Ma.Par.ParEBM;	//[8.4]
      A     #Motor.InManual;	//[8.4]
      O     #Ma.CmdOff;
      S     #Motor.CmdOff;
//  
      A     #Mon1.StTrue;
      O     #Mon1.StCtoFalse;
      ON    #Ma.Par.ParMon1IsLS;	//[6.1]
      ON    #Ma.Par.ParMon1StopByFault;
      A(;	//[6.0]
      O     #Mon1.StFalse;	//[6.0]
      O     #Mon1.StCtoTrue;	//[6.0]
      ON    #Ma.Par.ParMon1IsHL;	//[6.0]
      O     #Ma.InOverrideHLOutlet;	//[6.0]
      );
      ON    #Ma.Par.ParWithMon1;	//[7.4]
      A(;
      A     #Ma.Par.ParEBM;	//[7.6]
      O     #Mon2.StTrue;
      O     #Mon2.StCtoFalse;
      ON    #Ma.Par.ParMon2IsLS;
      );
      A(;
      A     #Ma.Par.ParEBM;	//[7.6]
      O     #Mon3.StTrue;
      O     #Mon3.StCtoFalse;
      ON    #Ma.Par.ParWithMon3;
      ON    #Ma.Par.ParMon3IsLS;
      );
      A(;
      A     #Ma.Par.ParEBM;	//[7.6]
      O     #Mon4.StTrue;	//[6.2]
      O     #Mon4.StCtoFalse;	//[6.2]
      A     #Ma.Par.ParMon4IsLS;	//[6.2]
      O(;	//[6.2]
      A     #Mon4.StFalse;	//[6.2]
      O     #Mon4.StCtoTrue;	//[6.2]
      O     #Ma.InOverrideHLOutlet;	//[6.2]
      AN    #Ma.Par.ParMon4IsLS;	//[6.2]
      );	//[6.2]
      ON    #Ma.Par.ParMon4StopByFault;	//[6.2]
      O     #Ma.Par.ParMon4IsSM;	//[8.0]
      ON    #Ma.Par.ParWithMon4;	//[6.2]
      );	//[6.2]
      A(;	//[7.0]
      A     #Ma.Par.ParEBM;	//[7.6]
      O     #Mon5.StTrue;	//[7.0]
      O     #Mon5.StCtoFalse;	//[7.0]
      ON    #Ma.Par.ParWithMon5;	//[7.0]
      );	//[7.0]
      A(;	//[7.0]
      A     #Ma.Par.ParEBM;	//[7.6]
      O     #Mon6.StTrue;	//[7.0]
      O     #Mon6.StCtoFalse;	//[7.0]
      ON    #Ma.Par.ParWithMon6;	//[7.0]
      );	//[7.0]
      =     #tmpEnable;	//[4.0]
//Set speed if manual mode without interlocking                   
      AN    #Motor.Par.ParManual;
      ON    #Ma.InManual;
      O     #Motor.InManual;
      JC    inJo;
      A     #Motor.InOutManSlow;
      =     #Motor.InSlow;
inJo: A(;
      AN    #Motor.Par.ParManual;
      AN    #Motor.InOutManRev;
      ON    #Ma.InManual;
      A     #Ma.InEnableFwd;
      O;
      A     #Ma.InManual;
      A     #Motor.Par.ParManual;
      AN    #Motor.InOutManRev;
      );
      AN    #Ma.InpLocked;
      AN    #tmpFaultStop;
      AN    #Ma.CmdOff;
      A     #tmpEnable;	//[4.0]
      =     #Motor.InEnableFwd;
      A(;
      AN    #Motor.Par.ParManual;
      A     #Motor.InOutManRev;
      ON    #Ma.InManual;
      A     #Ma.InEnableRev;
      O;
      A     #Ma.InManual;
      A     #Motor.Par.ParManual;
      A     #Motor.InOutManRev;
      );
      AN    #Ma.InpLocked;
      AN    #tmpFaultStop;
      AN    #Ma.CmdOff;
      A     #tmpEnable;	//[4.0]
      =     #Motor.InEnableRev;
      A     #Ma.CmdNext;
      AN    #Ma.InManual;
      O;
      A     #Ma.InManual;
      A     #Ma.CmdOn;
      S     #Motor.CmdNext;
      A     #Ma.InSeqStop;
      AN    #Ma.InManual;	// [3.1]
      =     #Motor.InSeqStop;
//--- Local mode --
      A     #Ma.InLocal;
      AN    #Ma.InManual;
      =     #tmpLocal;
      A     #tmpLocal;
      =     #Motor.InLocal;
      AN    #tmpFaultStop;	//[8.6]
      O     #tmpLocal;	//[8.6]
      AN    #Motor.InpRunFwd;	//[8.4]
      AN    #Motor.InpRunRev;	//[8.4]
      AN    #Motor.InManual;	//[8.4]
      A(;	//[8.6]
      L     #Motor.StCode;	//[8.6]
      L     0;	//[8.6]
      ==I;	//[8.6]
      O     #Motor.StStopped;	//[7.6]
      );	//[8.6]
      ON    #Ma.Par.ParEBM;	//[7.6]
      A     #tmpLocal;	//[7.6]
      =     #Mon4.InLocal;	//[7.6]
      AN    #tmpFaultStop;	//[8.6]
      O     #tmpLocal;	//[8.6]
      AN    #Motor.InpRunFwd;	//[8.4]
      AN    #Motor.InpRunRev;	//[8.4]
      AN    #Motor.InManual;	//[8.4]
      ON    #Ma.Par.ParEBM;	//[8.4]
      A     #tmpLocal;
      A(;	//[8.6]
      L     #Motor.StCode;	//[8.6]
      L     0;	//[8.6]
      ==I;	//[8.6]
      O     #Motor.StStopped;	//[7.6]
      );	//[8.6]
      =     #Mon1.InLocal;
      =     #Mon2.InLocal;
      =     #Mon3.InLocal;
      =     #Mon5.InLocal;	//[7.0]
      =     #Mon6.InLocal;	//[7.0]
//--- Monitoring
      A     #Ma.Par.ParMon1IsLS;
      O     #Motor.StStartedFwd;
      O     #Motor.StStartedRev;
      AN    #Ma.Par.ParMon1IsHL;
      =     #Mon1.InMonTrue;
      A     #Ma.Par.ParMon1IsHL;
      AN    #Ma.InOverrideHLOutlet;
      =     #Mon1.InMonFalse;
//Mon2
      A     #Ma.OutpFcttst_BM_Top;	//[7.0]
      =     #Mon2.InMonFalse;	//[7.0]
      A     #Ma.Par.ParMon2IsLS;
      O     #Motor.StStartedFwd;
      O     #Motor.StStartedRev;
      O     #Ma.Par.ParEBM;	//[7.3]
      AN    #Ma.OutpFcttst_BM_Bottom;	//[7.0]
      AN    #Mon2.InMonFalse;	//[7.0]
      =     #Mon2.InMonTrue;
//Mon3
      A     #Ma.OutpFcttst_BM_Top;	//[7.0]
      A     #Ma.Par.ParWithMon3;	//[7.0]
      =     #Mon3.InMonFalse;	//[7.0]
      A     #Ma.Par.ParMon3IsLS;
      O     #Motor.StStartedFwd;
      O     #Motor.StStartedRev;
      O     #Ma.Par.ParEBM;	//[7.3]
      AN    #Ma.OutpFcttst_BM_Bottom;	//[7.0]
      AN    #Mon3.InMonFalse;	//[7.0]
      =     #Mon3.InMonTrue;
//Mon4
      A     #Ma.Par.ParMon4AsWarning;	//[4.0]
      O     #Ma.Par.ParMon4IsLS;	//[5.0]
      O     #Ma.Par.ParEBM;	//[7.3]
      O(;	//[7.3]
      O     #Motor.StStartedFwd;	//[7.0]
      O     #Motor.StStartedRev;	//[7.0]
      A     #Ma.Par.ParMon4IsSM;	//[8.0]
      );	//[7.3]
      AN    #Ma.OutpFcttst_BM_Top;	//[7.0]
      AN    #Ma.OutpFcttst_BM_Bottom;	//[7.0]
      A     #Ma.Par.ParWithMon4;	//[7.0]
      =     #Mon4.InMonTrue;	//[4.0]
      A(;	//[8.0]
      AN    #Mon4.InMonTrue;	//[7.0]
      AN    #Ma.Par.ParEBM;	//[7.0]
      A     #Ma.Par.ParWithMon4;	//[7.0]
      O;
      A     #Ma.OutpFcttst_BM_Bottom;	//[7.0]
      A     #Ma.Par.ParWithMon4;	//[7.0]
      );	//[8.0]
      AN    #Ma.Par.ParMon4IsSM;	//[8.0]
      =     #Mon4.InMonFalse;
//Mon5
      A     #Ma.OutpFcttst_BM_Bottom;	//[7.0]
      A     #Ma.Par.ParWithMon5;	//[7.0]
      =     #Mon5.InMonFalse;	//[7.0]
      A     #Motor.StStartedFwd;	//[7.0]
      O     #Motor.StStartedRev;	//[7.0]
      O     #Ma.Par.ParEBM;	//[7.3]
      AN    #Ma.OutpFcttst_BM_Top;	//[7.0]
      AN    #Mon5.InMonFalse;	//[7.0]
      =     #Mon5.InMonTrue;	//[7.0]
//Mon6
      A     #Ma.OutpFcttst_SM;	//[7.0]
      A     #Ma.Par.ParWithMon6;	//[7.0]
      =     #Mon6.InMonFalse;	//[7.0]
      A     #Motor.StStartedFwd;	//[7.0]
      O     #Motor.StStartedRev;	//[7.0]
      O     #Ma.Par.ParEBM;	//[7.3]
      AN    #Mon6.InMonFalse;	//[7.0]
      =     #Mon6.InMonTrue;	//[7.0]
//--- Fault Reset -------------
      A     #Ma.CmdFaultReset;
      FP    #Ma.OutEdgeFaultReset;	//[8.3]
      S     #Mon4.CmdFaultReset;
      S     #Motor.CmdFaultReset;
      S     #Mon1.CmdFaultReset;
      S     #Mon2.CmdFaultReset;
      S     #Mon3.CmdFaultReset;
      S     #Mon5.CmdFaultReset;	//[7.0]
      S     #Mon6.CmdFaultReset;	//[7.0]
NETWORK
TITLE = Call Digital Input: Monitor B1
      AN    #Ma.Par.ParWithMon1;	//[7.0]
      JC    Mon2;	//[7.0]
      CALL  #Mon1;
NETWORK
TITLE = Call Digital Input: Monitor B2
Mon2: A     #Ma.InpControlEBM;	//[8.4]
      A     #Ma.OutpFcttst_BM_Top;	//[8.4]
      A     #Ma.Par.ParEBM;	//[8.4]
      O     #Mon2.InpTrue;	//[8.4]
      =     #Mon2.InpTrue;	//[8.4]
      CALL  #Mon2;
NETWORK
TITLE = Call Digital Input: Monitor B3
      AN    #Ma.Par.ParWithMon3;
      JC    Mon4;	//[7.0]
      A     #Ma.InpControlEBM;	//[8.4]
      A     #Ma.OutpFcttst_BM_Top;	//[8.4]
      A     #Ma.Par.ParEBM;	//[8.4]
      O     #Mon3.InpTrue;	//[8.4]
      =     #Mon3.InpTrue;	//[8.4]
      CALL  #Mon3;
NETWORK
TITLE = Call Digital Input: Mon4
Mon4: AN    #Ma.Par.ParWithMon4;	//[7.0]
      JC    Mon5;
      A     #Ma.InpControlEBM;	//[8.4]
      A     #Ma.OutpFcttst_BM_Bottom;	//[8.4]
      A     #Ma.Par.ParEBM;	//[8.4]
      O     #Mon4.InpTrue;	//[8.4]
      =     #Mon4.InpTrue;	//[8.4]
      CALL  #Mon4;
NETWORK
TITLE = Call Digital Input: Mon5  [7.0]
Mon5: AN    #Ma.Par.ParWithMon5;	//[7.0]
      JC    Mon6;	//[7.0]
      A     #Ma.InpControlEBM;	//[8.4]
      A     #Ma.OutpFcttst_BM_Bottom;	//[8.4]
      A     #Ma.Par.ParEBM;	//[8.4]
      O     #Mon5.InpTrue;	//[8.4]
      =     #Mon5.InpTrue;	//[8.4]
      CALL  #Mon5;	//[7.0]
NETWORK
TITLE = Call Digital Input: Mon6 [7.0]
Mon6: AN    #Ma.Par.ParWithMon6;	//[7.0]
      JC    Mo;	//[7.0]
      A     #Ma.InpControlEBM;	//[8.4]
      A     #Ma.OutpFcttst_SM;	//[8.4]
      A     #Ma.Par.ParEBM;	//[8.4]
      O     #Mon6.InpTrue;	//[8.4]
      =     #Mon6.InpTrue;	//[8.4]
      CALL  #Mon6;	//[7.0]
NETWORK
TITLE = Call Motor
Mo:   CALL  #Motor;
NETWORK
TITLE = State
// Stopped
      A(;	//[8.5]
      A     #Mon1.StTrue;	//[8.5]
      AN    #Ma.Par.ParMon1IsHL;	//[8.5]
      O;	//[8.5]
      A     #Mon1.StFalse;	//[8.5]
      A     #Ma.Par.ParMon1IsHL;	//[8.5]
      ON    #Ma.Par.ParMon1StopByFault;	//[8.5]
      ON    #Ma.Par.ParWithMon1;	//[8.5]
      );	//[8.5]
      A     #Mon2.StTrue;	//[8.5]
      A(;	//[8.5]
      A     #Mon3.StTrue;	//[8.5]
      ON    #Ma.Par.ParWithMon3;	//[8.5]
      );	//[8.5]
      A(;	//[8.5]
      A     #Ma.Par.ParMon4IsLS;	//[8.5]
      O     #Ma.Par.ParMon4IsSM;	//[8.5]
      A     #Mon4.StTrue;	//[8.5]
      O;	//[8.5]
      A     #Mon4.StFalse;	//[8.5]
      AN    #Ma.Par.ParMon4IsLS;	//[8.5]
      AN    #Ma.Par.ParMon4IsSM;	//[8.5]
      AN    #Ma.Par.ParEBM;	//[8.5]
      O     #Ma.Par.ParMon4AsWarning;	//[8.5]
      ON    #Ma.Par.ParMon4StopByFault;	//[8.5]
      ON    #Ma.Par.ParWithMon4;	//[8.5]
      );	//[8.5]
      A(;	//[8.5]
      A     #Mon5.StTrue;	//[8.5]
      ON    #Ma.Par.ParWithMon5;	//[8.5]
      );	//[8.5]
      A(;	//[8.5]
      A     #Mon6.StTrue;	//[8.5]
      ON    #Ma.Par.ParWithMon6;	//[8.5]
      );	//[8.5]
      =     #tmpMonElOk;	//[8.5]
// Stopped
      A     #Motor.StStopped;
      AN    #tmpFaultSum;
      AN    #Ma.InpLocked;
      =     #Ma.StStopped;
// Locked 
      A     #Motor.StStopped;
      AN    #tmpFaultSum;
      A     #Ma.InpLocked;
      =     #Ma.StLocked;
// Starting
      O     #Motor.StStartedFwd;	//[8.5]
      O     #Motor.StStartedRev;	//[8.5]
      AN    #tmpMonElOk;	//[8.5]
      AN    #Ma.StStartedFwd;	//[8.5]
      AN    #Ma.StStartedRev;	//[8.5]
      O     #Motor.StStarting;
      AN    #tmpFaultSum;
      =     #Ma.StStarting;
// StartedFwd
      A     #Motor.StStartedFwd;
      AN    #Ma.StStarting;	//[8.5]
      AN    #tmpFaultSum;
      =     #Ma.StStartedFwd;
// StartedRev
      A     #Motor.StStartedRev;
      AN    #Ma.StStarting;	//[8.5]
      AN    #tmpFaultSum;
      =     #Ma.StStartedRev;
// Stopping
      A     #Motor.StStopping;
      AN    #tmpFaultSum;
      =     #Ma.StStopping;
// Fault
      A     #tmpFaultSum;
      =     #Ma.StFault;
NETWORK
TITLE = Global End
      NOP   0;
//--------------------------------
//Pulse length OutpFaultReset is 500ms
      A     "GCS7_Gr_OutTick1s";	//[7.0]
      R     #Ma.OutpFaultReset;	//[7.0]
//--------------------------------
//Set OutpFaultReset
// - with tick  "GCS7_Gr_OutTick1s"
// - Negativ flag of Ma.InpControlEBM during test
      AN    #Ma.InpControlEBM;	//[7.6]
      A     #Ma.Par.ParEBM;	//[7.6]
      O     #Ma.StFault;	//[7.0]
      A     "GCS7_Gr_OutTick1s";	//[7.0]
      A     #Ma.CmdFaultReset;	//[7.0]
      O;
      A     #Ma.OutFaultResetFcttst;	//[7.5]
      AN    #Ma.StFault;	//[7.5]
      S     #Ma.OutpFaultReset;	//[7.0]
      R     #Ma.CmdFaultReset;	//[7.5]
      A     #Ma.OutpFaultReset;	//[7.5]
      A     #Ma.InpControlEBM;	//[7.6]
      R     #Ma.OutFaultResetFcttst;	//[7.5]
//--------------------------------
//Reset OutpFaultReset immediatly when InpControlEBM is ok
      A     #Ma.InpControlEBM;	//[7.6]
      O     #Ma.StFault;	//[7.6]
      A     #Ma.OutFaultResetFcttst;	//[7.5]
      R     #Ma.OutFaultResetFcttst;	//[7.5]
      R     #Ma.OutpFaultReset;	//[7.0]
//--------------------------------
//Reset  CmdFaultReset when no fault
      A     #Ma.InpControlEBM;	//[7.6]
      ON    #Ma.Par.ParEBM;	//[7.6]
      AN    #Ma.StFault;	//[7.0]
      R     #Ma.CmdFaultReset;	//[7.5]
//--------------------------------
//Init commands
      CLR;	//---Clear all commands
      =     #Ma.CmdOn;
      =     #Ma.CmdOff;
      =     #Ma.CmdNext;
NETWORK
TITLE = State Code
// Same as motor
      A     #Ma.StLocked;
      L     8;	//  StCode=Locked
      JC    Code;
      L     #Motor.StCode;	// StCode=Motor
      AN    #Ma.StFault;
      JC    Code;
      L     32;	// StCode=Fault
Code: L     #Ma.StCode;	// Old state code
      TAK;
      T     #Ma.StCode;	// Save state code
      <>I;
      L     3;
      CC    "SYS_CBitCtrl";	//Set change bit
END_FUNCTION_BLOCK

FUNCTION_BLOCK "GCS7_M_Motor2Mon"	// FB 51
TITLE = Motor with 2 monitoring elements
//  
//COPYRIGHT:    (C) 1997  BUHLER AG, CH-9240 UZWIL, SWITZERLAND
//
//PRODUCT:      GCS7
//
//TITLE:        FB 51 MACHINE-CONTROL:Motor with 2 Digital Input
//               
//-------------------------------------------------------------------------
//
//IDENT:        AUTHOR:             DEPT:                       DATE:
//
//FB51.4.2      A. Egli             CT3                         10-Apr-2008
//              - Interlocking check Ma.Par.ParWithMon1
//              - Init if download DB
//FB51.4.1      A. Egli             CT3                         14-Nov-2003
//              Interlocking check Ma.Par.ParWithMon2
//FB51.4.0      A. Egli             CT3                         17-Jun-2002
//              New Release with one block 
//FB51.3.4      A. Egli             CT3                         18-Oct-2001
//              Conditon for Prealarm with ParPS
//FB51.3.3      A. Egli             CT3                         26-Sep-2001
//              ParPS  GCPROVB: Revision 33
//FB51.3.2      A. Egli             CT3                         29-Jun-2001
//              ParManual 
//FB51.3.1      S. Kalberer         CT3                         10-Jan-2000
//              Set Mon1.InPreAlarmTrue instead of InPreAlarmFalse
//FB51.3.0      A. Egli             CT3                         11-Oct-1999
//              Local data reduced 
//FB51.2C       A. Egli             CT3                         03-Aug-1999
//              Test ParWithMon1 before call element
//FB51.2B       K. Tischer          MU664                       06-Mrz-1999
//              CC FC2 not UC FC2
//FB51.2A       A. Egli             CT3                         04-Mai-1998
//              StFault = StCode 32
//FB51.1A       A.Egli              AEE61                       5-Jul-1997
//              1st Release in S7
//
//-------------------------------------------------------------------------
//
//PURPOSE:      MANUAL : see [LL.M2IxxMAN]
//
//RESTRICTIONS: GCPROVB: Revision 33 for >=FB51.3.3
//              S7
//              ACCU2: Pointer to dynamic datas of the machine
//              ACCU1: Pointer to parameter datas of the machine
//
//-------------------------------------------------------------------------
//
AUTHOR : EA
FAMILY : GCS7LL
NAME : M_2DI
VERSION : 4.2
VAR
  Ma : UDT 20510;
  Mon1 : FB 14;	//Element
  Mon2 : FB 14;	//Element
  Motor : FB 12;	//Element
END_VAR
VAR_TEMP
  tmpFaultStop : BOOL ;
  tmpFaultSum : BOOL ;
  tmpLocal : BOOL ;
  tmpLenDyn : INT ;
  tmpEnable : BOOL ;
END_VAR
BEGIN
NETWORK
TITLE =
      L     10;
      T     #tmpLenDyn;
NETWORK
TITLE = PC Control
//=== Test Object number =====================
      L     "SYS_DirectCtrlDB".PC.ObjectNo;	//PCControl.ObjectNo
      L     #Ma.Par.ParObjectNo;	//Input ObjectNo
      <>I;
      JC    aEnd;
//=== Test OType      ========================
      L     2051;	//Input object type
      L     "SYS_DirectCtrlDB".PC.ObjectType;	//PCControl.ObjectType
      <>I;
      JC    aEnd;
//=== Test Handshake =========================
      A     "SYS_DirectCtrlDB".PC.Hsk.FExamine;	// Handshake.FExamine
      JC    aExa;
      A     "SYS_DirectCtrlDB".PC.Hsk.FDefineCmd;	// Handshake.FDefineCmd
      O     "SYS_DirectCtrlDB".PC.Hsk.FDefinePara;	// Handshake.FDefinePara
      JC    aCmd;
aIni: L     2;	// FcInit
      UC    "SYS_DirectCtrl";
      JU    aEnd;
// Write new commands from PC to Interface of group 
aCmd: A     "SYS_DirectCtrlDB".PC.Cmd1[8];	//Cmd1[8]=CmdOff
      S     #Ma.CmdOff;
      A     "SYS_DirectCtrlDB".PC.Cmd1[9];	//Cmd1[9]=CmdOn
      S     #Ma.CmdOn;
      A     "SYS_DirectCtrlDB".PC.Cmd1[10];	//Cmd1[10]=CmdNext
      S     #Ma.CmdNext;
      A     "SYS_DirectCtrlDB".PC.Cmd1[11];	//Cmd1[11]=CmdFaultReset
      S     #Ma.CmdFaultReset;
      A     "SYS_DirectCtrlDB".PC.Cmd1[13];	//Cmd1[13]=CmdManualOn
      S     #Ma.InManual;
      A     "SYS_DirectCtrlDB".PC.Cmd2[13];	//Cmd2[13]=CmdManualOff
      R     #Ma.InManual;
      A     "SYS_DirectCtrlDB".PC.Cmd1[6];	//Cmd1[14]=SlowOn
      S     #Motor.InOutManSlow;
      A     "SYS_DirectCtrlDB".PC.Cmd2[6];	//Cmd2[14]=SlowOff
      R     #Motor.InOutManSlow;
      A     "SYS_DirectCtrlDB".PC.Cmd1[7];	//Cmd1[15]=RevOn
      S     #Motor.InOutManRev;
      A     "SYS_DirectCtrlDB".PC.Cmd2[7];	//Cmd2[15]=RevOff
      R     #Motor.InOutManRev;
      AN    "SYS_DirectCtrlDB".PC.Hsk.FDefineCmd;	// Handshake.FDefineCmd
      JC    aIni;
      JU    aIni;
aExa: TAR2;	// Address Dynamic datas
      T     "SYS_DirectCtrlDB".GC.InDynAddr;	// -->PCControl.GC.InDynAddr
      L     #tmpLenDyn;	// Length Dynamic data
      T     "SYS_DirectCtrlDB".GC.InDynLen;	// -->PCControl.GC.InDynLen
      L     0;
      T     "SYS_DirectCtrlDB".GC.InParaAddr;	// -->PCControl.GC.InParaAddr
      T     "SYS_DirectCtrlDB".GC.InParaLen;	// -->PCControl.GC.InParaLen
      L     1;	// Code FcExamine
      UC    "SYS_DirectCtrl";
      L     10;	//Revision
      T     "SYS_DirectCtrlDB".GC.Revision;
aEnd: NOP   0;
NETWORK
TITLE = Interlocking
//===Global Group Orders===
      A     "GCS7_Gr_OutManualOn";	//Gr.OutManualOn
      S     #Ma.InManual;
      A     "GCS7_Gr_OutManualOff";	//Gr.OutManualOff
      R     #Ma.InManual;
      A     #Ma.InManual;
      S     "GCS7_Gr_InManual";	//Gr.InManual
      A     #Ma.InLocal;
      AN    #Ma.InManual;
      =     #tmpLocal;
//--- Fault----
      A     #Mon2.StFault;
      A     #Ma.Par.ParMon2StopByFault;
      O(;
      A     #Mon1.StFault;
      A     #Ma.Par.ParMon1StopByFault;
      );
      =     #tmpFaultStop;
      A     #Mon1.StFault;
      O     #Mon2.StFault;
      O     #Motor.StFault;
      =     #tmpFaultSum;
//--- Motor----
      A     #Mon1.StTrue;
      O     #Mon1.StCtoFalse;
      ON    #Ma.Par.ParMon1IsLS;
      ON    #Ma.Par.ParMon1StopByFault;
      ON    #Ma.Par.ParWithMon1;	//[4.2]
      A(;
      O     #Mon2.StTrue;
      O     #Mon2.StCtoFalse;
      ON    #Ma.Par.ParMon2IsLS;
      ON    #Ma.Par.ParMon2StopByFault;
      ON    #Ma.Par.ParWithMon2;	//[4.1]
      );
      =     #tmpEnable;	//[4.0]
      A(;	//3.2
      AN    #Motor.Par.ParManual;	//3.2
      AN    #Motor.InOutManRev;	//3.2
      ON    #Ma.InManual;	//3.2
      A     #Ma.InEnableFwd;	//3.2
      O;	//3.2
      A     #Ma.InManual;	//3.2
      A     #Motor.Par.ParManual;	//3.2
      AN    #Motor.InOutManRev;	//3.2
      );	//3.3
      AN    #tmpFaultStop;
      A     #tmpEnable;	//[6.0]
      AN    #Ma.CmdOff;
      =     #Motor.InEnableFwd;
      A(;	//3.2
      AN    #Motor.Par.ParManual;	//3.2
      A     #Motor.InOutManRev;	//3.2
      ON    #Ma.InManual;	//3.2
      A     #Ma.InEnableRev;	//3.2
      O;	//3.2
      A     #Ma.InManual;	//3.2
      A     #Motor.Par.ParManual;	//3.2
      A     #Motor.InOutManRev;	//3.2
      );	//3.2
      AN    #tmpFaultStop;
      AN    #Ma.CmdOff;
      A     #tmpEnable;	//[6.0]
      =     #Motor.InEnableRev;
      A     #Ma.CmdNext;
      AN    #Ma.InManual;
      O;
      A     #Ma.InManual;
      A     #Ma.CmdOn;
      S     #Motor.CmdNext;
      A     #Ma.InSeqStop;
      AN    #Ma.InManual;	//3.2
      =     #Motor.InSeqStop;
//--- Local mode --
      A     #tmpLocal;
      =     #Motor.InLocal;
      A(;	//[4.2]
      L     #Motor.StCode;	//[4.2]
      L     0;	//[4.2]
      ==I;	//[4.2]
      O     #Motor.StStopped;
      );	//[4.2]
      A     #tmpLocal;
      =     #Mon1.InLocal;
      A(;	//[4.2]
      L     #Motor.StCode;	//[4.2]
      L     0;	//[4.2]
      ==I;	//[4.2]
      O     #Motor.StStopped;
      );	//[4.2]
      O     #Ma.Par.ParMon2IsHL;
      A     #tmpLocal;
      O     #Ma.Par.ParMon2NoFault;
      =     #Mon2.InLocal;
//--- Monitoring
      O     #Motor.StStartedFwd;	//[3.3]
      O     #Motor.StStartedRev;	//[3.3]
      AN    #Mon1.InMonTrue;	//[3.3]
      A     #Ma.Par.ParMon1IsPS;	//[3.3]
      S     #Mon1.CmdRunTimeoutTime;	//[3.3]
      O     #Motor.StStartedFwd;
      O     #Motor.StStartedRev;
      O     #Ma.Par.ParMon1IsLS;
      =     #Mon1.InMonTrue;
      A     #Motor.StStartedFwd;
      O     #Motor.StStartedRev;
      AN    #Ma.Par.ParMon2IsHL;
      O     #Ma.Par.ParMon2IsLS;
      =     #Mon2.InMonTrue;
      A     #Ma.Par.ParMon2IsHL;
      =     #Mon2.InMonFalse;
      A     #Motor.StStartedFwd;	// [3.4]
      AN    #Mon1.OutTimeoutTime;	// [3.4]
      ON    #Ma.Par.ParMon1IsPS;	// [3.4]
      A     #Ma.Par.ParMon1PreAlarm;
      AN    #Mon1.CmdRunTimeoutTime;	// [3.4]
      =     #Mon1.InPreAlarmTrue;	//3.1: not InPreAlarmFalse
      AN    #Mon1.StTrue;
      A     #Mon1.InPreAlarmTrue;	// [3.4]
      A     #Ma.Par.ParWithMon1;	//[4.2]
      =     #Ma.OutWarning;
//--- Fault Reset -------------
      A     #Ma.CmdFaultReset;
      S     #Motor.CmdFaultReset;
      S     #Mon1.CmdFaultReset;
      S     #Mon2.CmdFaultReset;
NETWORK
TITLE = Set Mon1.OutDelayTime =0
      AN    #Motor.StStopped;	//[3.4  --->
      AN    #Motor.StFault;
      ON    #Mon1.StCtoFalse;
      ON    #Ma.Par.ParMon1IsPS;
      JC    Par0;
//Set Parameter
      L     0;
      T     #Mon1.Par.OutDelayTime;
Par0: NOP   0;	// <-- 3.4]
NETWORK
TITLE = Call Digital Input: Monitor B1
      AN    #Ma.Par.ParWithMon1;
      JC    B2;
      CALL  #Mon1;
NETWORK
TITLE = Call Digital Input: Monitor B2
B2:   AN    #Ma.Par.ParWithMon2;
      JC    Moto;
      CALL  #Mon2;
NETWORK
TITLE = Call Motor
Moto: CALL  #Motor;
NETWORK
TITLE = Jump to actual state
      A     #Ma.StStopped;
      JC    S0;	// ===> State
      A     #Ma.StStartedFwd;
      JC    S2;	// ===> State
      A     #Ma.StStarting;
      JC    S1;	// ===> State
      A     #Ma.StStopping;
      JC    S3;	// ===> State
      A     #Ma.StStartedRev;
      JC    S5;	// ===> State
      A     #Ma.StFault;
      JC    S4;	// ===> State
NETWORK
TITLE = Stopped
xxS0: S     #Ma.StStopped;
S0:   A     #tmpFaultSum;
      R     #Ma.StStopped;
      JC    xxS4;	//--> StFault
      AN    #Motor.StStopped;
      R     #Ma.StStopped;
      JC    xxS1;	//--> StStarting
      JU    OUT;
NETWORK
TITLE = Starting
xxS1: S     #Ma.StStarting;
S1:   A     #tmpFaultSum;
      R     #Ma.StStarting;
      JC    xxS4;	//--> StFault
// Condition for StStopping
      A     #Motor.StStopped;
      O     #Motor.StStopping;
      R     #Ma.StStarting;
      JC    xxS3;	//--> StStopping
      AN    #Mon1.StTrue;
      A     #Ma.Par.ParWithMon1;
      O;
      AN    #Mon2.StTrue;
      A     #Ma.Par.ParWithMon2;
      AN    #Ma.Par.ParMon2IsHL;
      JC    S2En;
// Condition for StStartedFwd
      A     #Motor.StStartedFwd;
      R     #Ma.StStarting;
      JC    xxS2;	//--> StStartedFwd
// Condition for StStartedFwd
      A     #Motor.StStartedRev;
      R     #Ma.StStarting;
      JC    xxS5;	//--> StStartedRev
S2En: JU    OUT;
NETWORK
TITLE = StartedFwd
xxS2: S     #Ma.StStartedFwd;
S2:   A     #tmpFaultSum;
      R     #Ma.StStartedFwd;
      JC    xxS4;	//--> StFault
// Condition for StStopping
      AN    #Motor.StStartedFwd;
      R     #Ma.StStartedFwd;
      JC    xxS3;	//--> StStopping
      JU    OUT;
NETWORK
TITLE = StartedRev
//any Transition 
xxS5: S     #Ma.StStartedRev;
//=== Logic
// Condition for StFault
S5:   A     #tmpFaultSum;
      R     #Ma.StStartedRev;
      JC    xxS4;	//--> StFault
// Condition for StStopping
      AN    #Motor.StStartedRev;
      R     #Ma.StStartedRev;
      JC    xxS3;	//--> StStopping
      JU    OUT;
NETWORK
TITLE = Stopping
xxS3: S     #Ma.StStopping;
S3:   A     #tmpFaultSum;
      R     #Ma.StStopping;
      JC    xxS4;	//--> StFault
// Condition for StStopped
      A     #Motor.StStopped;
      R     #Ma.StStopping;
      JC    xxS0;	//--> StStopped
// Condition for StStarting
      AN    #Motor.StStopping;
      R     #Ma.StStopping;
      JC    xxS1;	//--> StStarting
      JU    OUT;
NETWORK
TITLE = Fault
xxS4: S     #Ma.StFault;
S4:   AN    #tmpFaultSum;
      R     #Ma.StFault;
      JC    xxS3;	//--> StStopping
      JU    OUT;
NETWORK
TITLE = Global End
OUT:  CLR;	//---Clear all commands
      =     #Ma.CmdOn;
      =     #Ma.CmdOff;
      =     #Ma.CmdNext;
      =     #Ma.CmdFaultReset;
NETWORK
TITLE = State Code
// Same as motor
      L     32;	// StCode=Fault
      A     #Ma.StFault;
      JC    Code;
      L     2;	// StCode=Starting
      A     #Ma.StStarting;
      JC    Code;
      L     8;	// StCode=Warning
      A     #Ma.StStartedFwd;
      O     #Ma.StStartedRev;
      A     #Ma.OutWarning;
      JC    Code;
      L     #Motor.StCode;	// StCode=Motor
Code: L     #Ma.StCode;	// Old state code
      TAK;
      T     #Ma.StCode;	// Save state code
      <>I;
      L     3;
      CC    "SYS_CBitCtrl";	//Set change bit
END_FUNCTION_BLOCK

FUNCTION_BLOCK "GCS7_M_MotorBypass"	// FB 52
TITLE = Motor with bypass flap
//  
//COPYRIGHT:    (C) 1997  BUHLER AG, CH-9240 UZWIL,  SWITZERLAND
//
//PRODUCT:      GCS7
//
//TITLE:        FB 52 MACHINE-CONTROL:Motor with bypass flap
//              (GCPROVB Revision 11)
//-------------------------------------------------------------------------
//
//IDENT:        AUTHOR:             DEPT:                       DATE:
//FB52.6.2      A. Egli             CT3                         17-Jan-2007
//              Code: Revision set to 11
//FB52.6.1      A. Egli             CT3                         18-Feb-2006
//              InPressureOK
//FB52.6.0      A. Egli             CT3                         19-Oct-2005
//              Element Seal
//FB52.5.4      A. Egli             CT3                         26-Jan-2005
//              Transition StStopping --> StBypassed
//FB52.5.3      A. Egli             CT3                         11-Oct-2004
//              Restart Clearing time when changing position of bypass flap 
//FB52.5.2      A. Egli             CT3                         22-Apr-2004
//              For Clearing time check <=0 
//FB52.5.1      A. Egli             CT3                         26-Mai-2003
//              Condition StStarted, if Mon1 is HL
//              Send CmdOff to Motor
//FB52.5.0      A. Egli             CT3                         17-Jun-2002
//              New Release with one block 
//              If no Mon1 then reset ParMon1IsLS,ParMon1IsHL,ParMon1StopByFault
//FB52.4.1      A.Egli              CT3                         12-Mar-2002
//              InBypass2 
//FB52.4.0      A.Egli              CT3                         30-Jan-2002
//              VLS2: 2nd Bypass flap
//FB52.3.2      S. Kalberer         CT3                         09-Oct-2000
//              3.1 corrected and local mode for HLInlet if bypassed
//FB52.3.1      A. Egli             CT3                         08-Sep-2000
//              Local mode for motor if, bypassed
//FB52.3.0      A. Egli             CT3                         11-Oct-1999
//              Local data reduced 
//FB52.2C       A.Egli              CT3                         13-Sep-1999
//              Start condtion for motor by change maunal flap
//FB52.2B       K. Tischer          MU664                       06-Mrz-1999
//              CC FC2 not UC FC2
//FB52.2A       A. Egli             CT3                         04-Mai-1998
//              StFault = StCode 32
//FB52.1A       A.Egli              AEE61                       5-Jul-1997
//              1st Release in S7
//
//-------------------------------------------------------------------------
//
//PURPOSE:      MANUAL : see [LL.M1VxxMAN]
//
//RESTRICTIONS: S7
//              ACCU2: Pointer to dynamic datas of the machine
//              ACCU1: Pointer to parameter datas of the machine
//
//-------------------------------------------------------------------------
//
AUTHOR : EA
FAMILY : GCS7LL
NAME : M1V
VERSION : 6.3
VAR
  Ma : UDT 20520;
  Mon1 : FB 14;	//Element
  Motor : FB 12;	//Element
  VLS1 : FB 13;	//Element
  HLInlet : FB 14;	//Element
  VLS2 : FB 13;	//Element [4.0]
  Seal : FB 11;
END_VAR
VAR_TEMP
  tmpFaultSum : BOOL ;
  tmpLocal : BOOL ;
  tmpEnable : BOOL ;
  tmpStartReq : BOOL ;
  tmpLenDyn : INT ;
  tmpBypassed : BOOL ;
  StoreGrOutManualOff : BOOL ;
END_VAR
BEGIN
NETWORK
TITLE =
      L     16;
      T     #tmpLenDyn;
//Init flags
      AN    #Ma.Par.ParWithMon1;
      R     #Ma.Par.ParMon1IsLS;
      R     #Ma.Par.ParMon1IsHL;
      R     #Ma.Par.ParMon1StopByFault;
NETWORK
TITLE = PC Control
//=== Test Object number =====================
      L     "SYS_DirectCtrlDB".PC.ObjectNo;	//PCControl.ObjectNo
      L     #Ma.Par.ParObjectNo;	//Input ObjectNo
      <>I;
      JC    aEnd;
//=== Test OType      ========================
      L     2052;	//Input object type
      L     "SYS_DirectCtrlDB".PC.ObjectType;	//PCControl.ObjectType
      <>I;
      JC    aEnd;
//=== Test Handshake =========================
      A     "SYS_DirectCtrlDB".PC.Hsk.FExamine;	// Handshake.FExamine
      JC    aExa;
      A     "SYS_DirectCtrlDB".PC.Hsk.FDefineCmd;	// Handshake.FDefineCmd
      JC    aCmd;
      A     "SYS_DirectCtrlDB".PC.Hsk.FDefinePara;	// Handshake.FDefinePara
      JC    pPar;
aIni: L     2;	// FcInit
      UC    "SYS_DirectCtrl";
      JU    aEnd;
// Write parameter 
pPar: LAR1  P#DBX 58.0;
      L     P#6.0;
      +AR1;
      L     DBW [AR1,P#4.0];
      T     #Ma.Par.ParClearingTime;
// Write new commands from PC to Interface of group 
aCmd: A     "SYS_DirectCtrlDB".PC.Cmd1[8];	//Cmd1[8]=CmdOff
      S     #Ma.CmdOff;
      A     "SYS_DirectCtrlDB".PC.Cmd1[9];	//Cmd1[9]=CmdOn
      S     #Ma.CmdOn;
      A     "SYS_DirectCtrlDB".PC.Cmd1[10];	//Cmd1[10]=CmdNext
      S     #Ma.CmdNext;
      A     "SYS_DirectCtrlDB".PC.Cmd1[11];	//Cmd1[11]=CmdFaultReset
      S     #Ma.CmdFaultReset;
      A     "SYS_DirectCtrlDB".PC.Cmd1[13];	//Cmd1[13]=CmdManualOn
      S     #Ma.InManual;
      A     "SYS_DirectCtrlDB".PC.Cmd2[13];	//Cmd2[13]=CmdManualOff
      R     #Ma.InManual;
      R     #Motor.InManual;
      R     #VLS1.InManual;
      R     #VLS2.InManual;	//[4.0]
      A     "SYS_DirectCtrlDB".PC.Cmd1[5];	//Cmd1[5]=CmdBypass
      S     #Ma.InBypass;	//[6.0]
      S     #Ma.InBypass2;	//[6.0]
      A     "SYS_DirectCtrlDB".PC.Cmd2[5];	//Cmd1[5]=CmdMachine
      R     #Ma.InBypass;	//[6.0]
      R     #Ma.InBypass2;	//[6.0]
      S     #Ma.CmdOn;	//[6.0]
      JU    aIni;
aExa: TAR2;	// Address dynamic data
      T     "SYS_DirectCtrlDB".GC.InDynAddr;	// -->PCControl.GC.InDynAddr
      L     #tmpLenDyn;	// Length Dynamic data
      T     "SYS_DirectCtrlDB".GC.InDynLen;	// -->PCControl.GC.InDynLen
      L     0;
      T     "SYS_DirectCtrlDB".GC.InParaAddr;	// -->PCControl.GC.InParaAddr
      T     "SYS_DirectCtrlDB".GC.InParaLen;	// -->PCControl.GC.InParaLen
      L     1;	// Code FcExamine
      UC    "SYS_DirectCtrl";
      L     11;	//Revision
      T     "SYS_DirectCtrlDB".GC.Revision;
aEnd: NOP   0;
NETWORK
TITLE = Interlocking
//===Global Group Orders===
      A     "GCS7_Gr_OutManualOn";	//Gr.OutManualOn
      S     #Ma.InManual;
      A     "GCS7_Gr_OutManualOff";	//Gr.OutManualOff
      R     #Ma.InManual;
      A     #Ma.InManual;
      S     "GCS7_Gr_InManual";	//Gr.InManual
      A     #Ma.InLocal;
      AN    #Ma.InManual;
      =     #tmpLocal;
//--Bypassed ---------------
      A     #Ma.InBypass2;	//[6.3]
      O     #Ma.Par.ParLocalPosition;	//[6.3]
      A     #VLS2.StHN;	//[6.3]
      ON    #Ma.Par.ParWithVLS2;	//[6.3]
      A     #VLS1.StHN;	//[6.3]
      A(;	//[6.3]
      A     #Ma.InBypass;	//[6.3]
      O     #Ma.Par.ParLocalPosition;	//[6.3]
      );	//[6.3]
      =     #tmpBypassed;	//[6.3]
//--- Fault----
      A     #VLS2.StFault;	//[4.0]
      A     #Ma.Par.ParWithVLS2;	//[4.0]
      O     #Mon1.StFault;
      O;
      A     #Motor.StFault;
      AN    #tmpBypassed;	//[6.3]
      O     #VLS1.StFault;
      O     #HLInlet.StFault;
      =     #tmpFaultSum;
//---Interlocking
      A(;
      O     #VLS2.StLN;	//[4.0]
      O     #VLS2.StCtoLN;	//[4.0]
      A     #Ma.Par.ParWithVLS2;	//[4.0]
      O     #VLS1.StLN;
      O     #VLS1.StCtoLN;	//[2C]
      A     #Ma.Par.ParLocalPosition;
      O;
      A(;
      AN    #Ma.InBypass2;	//[4.0]
      A     #Ma.Par.ParWithVLS2;	//[4.0]
      ON    #Ma.InBypass;
      );
      AN    #Ma.Par.ParLocalPosition;
      );
//[6.0]      UN    #Ma.InManual
      AN    #tmpLocal;
      =     #tmpStartReq;
      A     #Mon1.StTrue;
      ON    #Ma.Par.ParMon1IsLS;
      AN    #Mon1.StFault;
      ON    #Ma.Par.ParMon1StopByFault;
      AN    #Ma.CmdOff;
      A(;
      A     #tmpStartReq;
      ON    #Ma.StBypassed;
//[6.0] O     #Ma.InManual
      );
      =     #tmpEnable;
//---Seal----
//[6.0] --->
      A     #Ma.CmdNext;
      AN    #Ma.InManual;
      A     #tmpStartReq;
      O;
      A     #Ma.CmdOn;
      A     #Ma.InManual;
      A     #tmpStartReq;
      S     #Seal.CmdNext;
      SET;
      =     #Seal.InEnable;
      A     #Seal.StStopped;
      A     #Motor.InLocal;
      AN    #tmpStartReq;
      O     #tmpLocal;
      =     #Seal.InLocal;
      A     #Seal.StStarted;
      A     #Motor.StStopped;
      S     #Seal.InSeqStop;
      A     #Ma.InEnableFwd;
      O     #Ma.InEnableRev;
      O     #Ma.CmdOn;
      A     #tmpEnable;
      A     #Ma.InPressureOK;	//[6.1]
      A     #tmpStartReq;
      R     #Seal.InSeqStop;
//<---[6.0]
//--- Motor----
      A     #Ma.CmdOff;	//[5.1]
      S     #Motor.CmdOff;	//[5.1]
      A     #tmpStartReq;
      AN    #Motor.StStartedFwd;
      AN    #Motor.StStartedRev;
      A(;	//[6.0]
      A     #Seal.StStarted;	//[6.0]
      A     #Ma.InPressureOK;	//[6.1]
      ON    #Ma.Par.ParWithSeal;	//[6.0]
      );	//[6.0]
      =     #Ma.OutStartReq;
      A     #tmpEnable;	//[6.0]
      A(;	//[6.0]
      A     #Seal.StStarted;	//[6.0]
      A     #Ma.InPressureOK;	//[6.1]
      ON    #Ma.Par.ParWithSeal;	//[6.0]
      );	//[6.0]
      =     #tmpEnable;	//[6.0]
      A     #Ma.InManual;	//[6.0]
      A     #Motor.Par.ParManual;	//[6.0]
      O     #Ma.InEnableFwd;
      A     #tmpEnable;
      =     #Motor.InEnableFwd;
      A     #tmpEnable;
      A     #Ma.InEnableRev;
      =     #Motor.InEnableRev;
      A     #Ma.OutStartReq;
      AN    #Ma.InManual;
      A     #Ma.CmdNext;
      O;
      A     #Ma.InManual;
      A     #Ma.CmdOn;
      S     #Motor.CmdNext;
      AN    #Seal.StStarted;	//[6.1]
      ON    #Ma.InPressureOK;	//[6.1]
      A     #Ma.Par.ParWithSeal;	//[6.1]
      S     #Motor.CmdOff;	//[6.1]
      A     #Ma.InSeqStop;
      AN    #Ma.InManual;	//[6.0]
      =     #Motor.InSeqStop;
//--- VLS----
      A     #Ma.InBypass;
      AN    #Ma.Par.ParLocalPosition;
      =     #VLS1.InEnableHN;
      A     #Motor.StStartedFwd;
      O     #Motor.StStartedRev;
      AN    #Ma.InBypass;
      AN    #Ma.Par.ParLocalPosition;
      =     #VLS1.InEnableLN;
      A     #Ma.InBypass2;
      AN    #Ma.Par.ParLocalPosition;
      =     #VLS2.InEnableHN;	//[4.0]
      A     #Motor.StStartedFwd;
      O     #Motor.StStartedRev;
      AN    #Ma.InBypass2;
      AN    #Ma.Par.ParLocalPosition;
      =     #VLS2.InEnableLN;	//[4.0]
      SET;
      S     #VLS1.CmdNext;
      S     #VLS2.CmdNext;	//[4.0]
//--- Local mode --
      A     #tmpLocal;
      =     #VLS1.InLocal;
      =     #VLS2.InLocal;	//[4.0]
      A     #VLS2.StHN;	//[4.0]
      AN    #VLS2.InEnableLN;	//[4.0]
      ON    #Ma.Par.ParWithVLS2;	//[4.0]
      A     #VLS1.StHN;	//[3.2 -->
      AN    #VLS1.InEnableLN;
      O     #tmpLocal;
      =     #HLInlet.InLocal;
      A     #VLS2.StHN;	//[4.0]
      ON    #Ma.Par.ParWithVLS2;	//[4.0]
      A     #VLS1.StHN;
      A     #Motor.StStopped;
      O     #tmpLocal;
      S     #Motor.InLocal;
      A(;
      AN    #Ma.InBypass2;	//[4.0]
      A     #Ma.Par.ParWithVLS2;	//[4.0]
      ON    #Ma.InBypass;
      AN    #Ma.Par.ParLocalPosition;
      O;
      AN    #VLS1.StHN;
      A     #Ma.Par.ParLocalPosition;
      O;
      AN    #VLS2.StHN;	//[4.0]
      A     #Ma.Par.ParLocalPosition;	//[4.0]
      A     #Ma.Par.ParWithVLS2;	//[4.0]
      );
      AN    #tmpLocal;
      R     #Motor.InLocal;	// <-- 3.2]
//      UN    #Ma.InBypass;  //[3.1 -->
//      UN    #Ma.Par.ParLocalPosition;
//      ON    #VLS.InEnableHN;
//      UN    #tmpLocal; 
//      R     #Motor.InLocal;
//      U     #VLS.InEnableHN;
//      U     #Motor.StStopped;
//      O     #tmpLocal; 
//      S     #Motor.InLocal; // <-- 3.1]
      A     #Motor.StStopped;
      ON    #Ma.Par.ParMon1IsLS;
      A     #tmpLocal;
      =     #Mon1.InLocal;
//--- Monitoring
      A     #Motor.StStartedFwd;
      O     #Motor.StStartedRev;
      AN    #Ma.Par.ParMon1IsHL;
      O(;
      AN    #VLS2.StHN;	//[4.0]
      A     #Ma.Par.ParWithVLS2;	//[4.0]
      O     #Ma.OutStartReq;
      ON    #Motor.StStopped;
      ON    #VLS1.StHN;
      A     #Ma.Par.ParMon1IsLS;
      );
      =     #Mon1.InMonTrue;
      A     #Ma.Par.ParMon1IsHL;
      =     #Mon1.InMonFalse;
      SET;
      =     #HLInlet.InMonFalse;
//--- Fault Reset -------------
      A     #Ma.CmdFaultReset;
      S     #Mon1.CmdFaultReset;
      S     #Motor.CmdFaultReset;
      S     #VLS1.CmdFaultReset;
      S     #HLInlet.CmdFaultReset;
      S     #VLS2.CmdFaultReset;	//[4.0]
      S     #Seal.CmdFaultReset;	//[6.0]
NETWORK
TITLE = Call Digital Input: Monitor B1
      AN    #Ma.Par.ParWithMon1;
      JC    Moto;
      CALL  #Mon1;
NETWORK
TITLE = Call Motor / Seal
Moto: A     "GCS7_Gr_OutManualOff";	//[6.3]
      =     #StoreGrOutManualOff;	//[6.3]
      A     #tmpBypassed;	//[6.3]
      AN    #Ma.InLocal;	//[6.3]
      R     "GCS7_Gr_OutManualOff";	//[6.3]
//Call Motor
      CALL  #Motor;
//Call Seal
      AN    #Ma.Par.ParWithSeal;
      JC    mot2;
      CALL  #Seal;
mot2: A     #StoreGrOutManualOff;	//[6.3]
      =     "GCS7_Gr_OutManualOff";	//[6.3] 
NETWORK
TITLE = Call VLS1
      CALL  #VLS1;
NETWORK
TITLE = Call VLS2
      AN    #Ma.Par.ParWithVLS2;
      JC    elHL;
      CALL  #VLS2;
NETWORK
TITLE = Call Digital Input: HL Inlet
elHL: AN    #Ma.Par.ParWithHLInlet;
      JC    StJ0;
      CALL  #HLInlet;
NETWORK
TITLE = Jump to actual state
StJ0: A     #Ma.StStopped;
      JC    S0;	// ===> State
      A     #Ma.StStarted;
      JC    S2;	// ===> State
      A     #Ma.StStarting;
      JC    S1;	// ===> State
      A     #Ma.StStopping;
      JC    S3;	// ===> State
      A     #Ma.StClearing;
      JC    S5;	// ===> State
      A     #Ma.StBypassed;
      JC    S6;	// ===> State
      A     #Ma.StFault;
      JC    S4;	// ===> State
NETWORK
TITLE = Stopped
xxS0: S     #Ma.StStopped;
S0:   A     #tmpFaultSum;
      R     #Ma.StStopped;
      JC    xxS4;	//--> StFault
      AN    #Motor.StStopped;
      R     #Ma.StStopped;
      JC    xxS1;	//--> StStarting
// Condition for StBypassed
      A     #VLS2.StHN;	// Bypassed [4.0]
      ON    #Ma.Par.ParWithVLS2;	//[4.0]
      A     #VLS1.StHN;	// Bypassed
      R     #Ma.StStopped;
      JC    xxS6;	//--> StBypassed
      JU    OUT;
NETWORK
TITLE = Starting
xxS1: S     #Ma.StStarting;
S1:   A     #tmpFaultSum;
      R     #Ma.StStarting;
      JC    xxS4;	//--> StFault
// Condition for StStopping
      A     #Motor.StStopped;
      O     #Motor.StStopping;
      R     #Ma.StStarting;
      JC    xxS3;	//--> StStopping
// Condition for StStarted
      A     #Mon1.StTrue;
      ON    #Ma.Par.ParWithMon1;
      O     #Ma.Par.ParMon1IsHL;	//5.1
      A(;
      O     #Motor.StStartedFwd;
      O     #Motor.StStartedRev;
      );
      R     #Ma.StStarting;
      JC    xxS2;	//--> StStarted
// Condition for StBypassed
      A     #VLS2.StHN;	//[6.3]
      ON    #Ma.Par.ParWithVLS2;	//[6.3]
      A     #VLS1.StHN;	//[6.3]
      R     #Ma.StStarting;	//  [6.3]
      JC    xxS6;	//--> StBypassed
      JU    OUT;
NETWORK
TITLE = Started
xxS2: S     #Ma.StStarted;
S2:   A     #tmpFaultSum;
      R     #Ma.StStarted;
      JC    xxS4;	//--> StFault
// Condition for StStopping
      AN    #Motor.StStartedRev;
      AN    #Motor.StStartedFwd;
      R     #Ma.StStarted;
      JC    xxS3;	//--> StStopping
// Condition for StClearing
      A     #VLS2.StHN;	//[4.0]
      ON    #Ma.Par.ParWithVLS2;	//[4.0]
      A     #VLS1.StHN;
      R     #Ma.StStarted;
      JC    xxS5;	//--> StClearing
      JU    OUT;
NETWORK
TITLE = StClearing
//any Transition 
xxS5: S     #Ma.StClearing;
      L     #Ma.Par.ParClearingTime;
      T     #Ma.Par.OutClearingTime;
//=== Logic
// Condition for StFault
S5:   A     #tmpFaultSum;
      R     #Ma.StClearing;
      JC    xxS4;	//--> StFault
// Condition for StStarted
      A     #Motor.StStartedFwd;
      O     #Motor.StStartedRev;
      A     #VLS1.StLN;
      A(;	//[4.0]
      A     #VLS2.StLN;	//[4.0]
      ON    #Ma.Par.ParWithVLS2;	//[4.0]
      );
      R     #Ma.StClearing;
      JC    xxS2;	//--> StStarted
      A     #VLS2.StHN;	//[5.3]
      ON    #Ma.Par.ParWithVLS2;	//[5.3]
      A     #VLS1.StHN;	//[5.3]
      JC    S5J1;	//[5.3]
      L     #Ma.Par.ParClearingTime;	//[5.3]
      T     #Ma.Par.OutClearingTime;	//[5.3]
S5J1: NOP   0;	//[5.3]
// Condition for StBypassed
      L     0;
      L     #Ma.Par.OutClearingTime;
      >=I;	//[5.2]
      R     #Ma.StClearing;
      JC    xxS6;	//--> StBypassed
// Condition for StStopping
      AN    #Motor.StStartedFwd;
      AN    #Motor.StStartedRev;
      R     #Ma.StClearing;
      JC    xxS3;	//--> StStopping
      ON    "GCS7_Gr_OutTick500ms";	//Gr.OutTick500ms
      JC    OUT;
      L     #Ma.Par.OutClearingTime;
      +     -5;
      T     #Ma.Par.OutClearingTime;
      JU    OUT;
NETWORK
TITLE = StBypassed
//any Transition 
xxS6: S     #Ma.StBypassed;
//=== Logic
// Condition for StFault
S6:   A     #tmpFaultSum;
      R     #Ma.StBypassed;
      JC    xxS4;	//--> StFault
// Condition for StStarted
      A     #Motor.StStartedFwd;
      O     #Motor.StStartedRev;
      AN    #VLS1.StHN;
      A(;	//[4.0]
      AN    #VLS2.StHN;	//[4.0]
      ON    #Ma.Par.ParWithVLS2;	//[4.0]
      );	//[4.0]
      R     #Ma.StBypassed;
      JC    xxS2;	//--> StStarted
// Condition for StStopping
      AN    #VLS1.StHN;	// Bypassed
      AN    #VLS1.StCtoLN;	//[2C]
      O(;	//[4.0]
      AN    #VLS2.StHN;	//[4.0]
      AN    #VLS2.StCtoLN;	//[4.0]
      A     #Ma.Par.ParWithVLS2;	//[4.0]
      );	//[4.0]
      R     #Ma.StBypassed;
      JC    xxS3;	//--> StStopping
      JU    OUT;
NETWORK
TITLE = Stopping
xxS3: S     #Ma.StStopping;
S3:   A     #tmpFaultSum;
      R     #Ma.StStopping;
      JC    xxS4;	//--> StFault
// Condition for StStopped
      A     #Motor.StStopped;
      R     #Ma.StStopping;
      JC    xxS0;	//--> StStopped
// Condition for StStarting
      AN    #Motor.StStopping;
      R     #Ma.StStopping;
      JC    xxS1;	//--> StStarting
// Condition for StBypassed
      A     #VLS2.StHN;	//[5.4] Bypassed
      ON    #Ma.Par.ParWithVLS2;	//[5.4]
      A     #VLS1.StHN;	//[5.4] Bypassed
      R     #Ma.StStopping;	//[5.4]
      JC    xxS6;	//[5.4]--> StBypassed
      JU    OUT;
NETWORK
TITLE = Fault
xxS4: S     #Ma.StFault;
S4:   AN    #tmpFaultSum;
      R     #Ma.StFault;
      JC    xxS3;	//--> StStopping
      JU    OUT;
NETWORK
TITLE = Global End
//---Clear all commands
OUT:  AN    #Seal.StStarting;	//[6.0]
      AN    #Seal.StStarted;	//[6.0]
      O     #Ma.OutStartReq;	//[6.0]
      O     #Ma.StFault;	//[6.0]
      ON    #Ma.InManual;	//[6.0]
      O     #Ma.CmdOff;	//[6.0]
      R     #Ma.CmdOn;
      CLR;
      =     #Ma.CmdOff;
      =     #Ma.CmdNext;
      =     #Ma.CmdFaultReset;
NETWORK
TITLE = State Code
// Same as motor
      L     32;	// StCode=Fault
      A     #Ma.StFault;
      JC    Code;
      L     8;	// StCode=Clearing
      A     #Ma.StClearing;
      JC    Code;
      L     9;	// StCode=ByPassed
      A     #Ma.StBypassed;
      JC    Code;
      L     1;	// StCode=Stopped  //[6.0]
      A     #Ma.StStopped;	//[6.0]
      JC    Code;	//[6.0]
      L     #Motor.StCode;	// StCode=Motor
Code: L     #Ma.StCode;	// Old state code
      TAK;
      T     #Ma.StCode;	// Save state code
      <>I;
      L     3;
      CC    "SYS_CBitCtrl";	//Set change bit
END_FUNCTION_BLOCK

FUNCTION_BLOCK "GCS7_M_Hopper"	// FB 53
TITLE = Hopper with 3 VLS and 1 DO
//  
//COPYRIGHT:    (C) 1997  BUHLER AG, CH-9240 UZWIL, SWITZERLAND
//
//PRODUCT:      GCS7
//
//TITLE:        FB 53 Machine Hopper: 3 Valve + digital output or motor
//
//-------------------------------------------------------------------------
//
//IDENT:        AUTHOR:             DEPT:                       DATE:
//
//FB53.6.2      A. Egli             CT3                         21-Mai-2007
//              InDisable Vibro
//FB53.6.1      A. Egli             CT3                         17-Jun-2002
//              OutDisableRead also for VLSUpper.Par.ParContValve
//FB53.6.0      A. Egli             CT3                         17-Jun-2002
//              New Release with one block 
//              Update to Version 5.3
//FB53.5.2      A.Egli              CT3                         31-Jan-2002
//              Init #Ma.OutPulseClose in State StClosed
//FB53.5.1      A.Egli              CT3                         19-Oct-2001
//              Condition for closing, if only VLSUpper is used
//FB53.5.0      K. Tischer          CT3                         01-Jun-2001
//              Optional VLSAirflap2 adapted
//FB53.4.1      S. Kalberer         CT3                         22-Nov-2000
//              Optional VLSLower adapted
//FB53.4.0      A. Egli             CT3                         24-Mai-2000
//              Type of Vibro is FB11 or FB12 
//FB53.3.0      A. Egli             CT3                         11-Oct-1999
//              Local data reduced 
//FB53.2B       K. Tischer          MU664                       06-Mrz-1999
//              CC FC2 not UC FC2
//FB53.2A       A. Egli             CT3                         04-Mai-1998
//              StFault = StCode 32
//FB53.1A       A.Egli              AEE61                       5-Jul-1997
//              1st Release in S7
//
//-------------------------------------------------------------------------
//
//PURPOSE:      MANUAL : see [LL.HOPxxMAN]
//
//RESTRICTIONS: S7
//              ACCU2: Pointer to dynamic datas of the machine
//              ACCU1: Pointer to parameter datas of the machine
//
//-------------------------------------------------------------------------
//
AUTHOR : EA
FAMILY : GCS7LL
NAME : Hopper
VERSION : 6.2
VAR
  Ma : UDT 20530;
  AirFlap : FB 13;	//Element
  VLSLower : FB 13;	//Element
  VLSUpper : FB 13;	//Element
  Vibro : FB 12;	//Element
  AirFlap2 : FB 13;	//Element [5.0]
END_VAR
VAR_TEMP
  tmpFaultSum : BOOL ;
  tmpLocal : BOOL ;
  tmpOpenReq : BOOL ;
  tmpLenDyn : INT ;
  tmpStoreAR2 : DINT ;
END_VAR
BEGIN
NETWORK
TITLE =
      L     16;
      T     #tmpLenDyn;
NETWORK
TITLE = PC Control
      NOP   0;
//=== Test Object number =====================
      L     "SYS_DirectCtrlDB".PC.ObjectNo;	//PCControl.ObjectNo
      L     #Ma.Par.ParObjectNo;	//Input ObjectNo
      <>I;
      JC    aEnd;
//=== Test OType      ========================
      L     2053;	//Input object type
      L     "SYS_DirectCtrlDB".PC.ObjectType;	//PCControl.ObjectType
      <>I;
      JC    aEnd;
//=== Test Handshake =========================
      A     "SYS_DirectCtrlDB".PC.Hsk.FExamine;	// Handshake.FExamine
      JC    aExa;
      A     "SYS_DirectCtrlDB".PC.Hsk.FDefineCmd;	// Handshake.FDefineCmd
      JC    aCmd;
      A     "SYS_DirectCtrlDB".PC.Hsk.FDefinePara;	// Handshake.FDefinePara
      JC    pPar;
aIni: L     2;	// FcInit
      UC    "SYS_DirectCtrl";
      JU    aEnd;
// Write parameter 
pPar: LAR1  P#DBX 58.0;
      L     P#6.0;
      +AR1;
      L     DBW [AR1,P#4.0];
      T     #Ma.Par.ParPulseClosing;
      L     DBW [AR1,P#6.0];
      T     #Ma.Par.ParWaitOpen;
// Write new commands from PC to Interface of group 
aCmd: A     "SYS_DirectCtrlDB".PC.Cmd1[8];	//Cmd1[8]=CmdClose
      S     #Ma.CmdClose;
      A     "SYS_DirectCtrlDB".PC.Cmd1[9];	//Cmd1[9]=CmdOpen
      S     #Ma.CmdOpen;
      A     "SYS_DirectCtrlDB".PC.Cmd1[9];	//Cmd1[10]=CmdNext
      S     #Ma.CmdNext;	//[6.0]
      A     "SYS_DirectCtrlDB".PC.Cmd1[11];	//Cmd1[11]=CmdFaultReset
      S     #Ma.CmdFaultReset;
      A     "SYS_DirectCtrlDB".PC.Cmd1[13];	//Cmd1[13]=CmdManualOn
      S     #Ma.InManual;
      A     "SYS_DirectCtrlDB".PC.Cmd2[13];	//Cmd2[13]=CmdManualOff
      R     #Ma.InManual;
      R     #AirFlap.InManual;
      R     #VLSUpper.InManual;
      R     #VLSLower.InManual;
      R     #Vibro.InManual;
      R     #AirFlap2.InManual;	//[5.0]
      JU    aIni;
aExa: TAR2;	// Address dynamic data
      T     "SYS_DirectCtrlDB".GC.InDynAddr;	// -->PCControl.GC.InDynAddr
      L     #tmpLenDyn;	// Length Dynamic data
      T     "SYS_DirectCtrlDB".GC.InDynLen;	// -->PCControl.GC.InDynLen
      L     0;
      T     "SYS_DirectCtrlDB".GC.InParaAddr;	// -->PCControl.GC.InParaAddr
      T     "SYS_DirectCtrlDB".GC.InParaLen;	// -->PCControl.GC.InParaLen
      L     1;	// Code FcExamine
      UC    "SYS_DirectCtrl";
      L     10;	//Revision
      T     "SYS_DirectCtrlDB".GC.Revision;
aEnd: NOP   0;
NETWORK
TITLE = Interlocking
      NOP   0;
//===Global Group Orders===
      A     "GCS7_Gr_OutManualOn";	//Gr.OutManualOn
      S     #Ma.InManual;
      A     "GCS7_Gr_OutManualOff";	//Gr.OutManualOff
      R     #Ma.InManual;
      A     #Ma.InManual;
      S     "GCS7_Gr_InManual";	//Gr.InManual
      A     #Ma.InLocal;
      AN    #Ma.InManual;
      =     #tmpLocal;
      A     #Ma.CmdOpen;
      S     #Ma.OutOpenManReq;
      A     #Ma.CmdClose;
      ON    #Ma.InManual;
      R     #Ma.OutOpenManReq;
//--- Fault----
      A     #AirFlap.StFault;
      O     #VLSLower.StFault;
      O     #VLSUpper.StFault;
      O     #Vibro.StFault;
      O     #AirFlap2.StFault;	//[5.0]
      =     #tmpFaultSum;
//--- Sequence opening ----
      A     #Ma.OutOpenManReq;
      A     #Ma.InManual;
      O;
      A     #Ma.InEnableOpen;
      AN    #AirFlap.StFault;	//[5.0] by fault airflap close
      AN    #AirFlap2.StFault;	//[5.0] by fault airflap close
      AN    #Ma.InManual;
      AN    #tmpLocal;
      =     #tmpOpenReq;
      A     #tmpOpenReq;
      S     #AirFlap.InEnableHN;
      S     #AirFlap2.InEnableHN;	//[5.0]
      A     #AirFlap.StHN;
      ON    #Ma.Par.ParWithAirFlap;
      A(;	//[5.0]
      A     #AirFlap2.StHN;	//[5.0]
      ON    #Ma.Par.ParWithAirFlap2;	//[5.0]
      );	//[5.0]
      A     #tmpOpenReq;
      S     #VLSLower.InEnableHN;
      AN    #Ma.OutPulseClose;
      ON    #Ma.Par.ParPulsing;
      A     #tmpOpenReq;
      A(;	//[4.1->]
      AN    #Ma.Par.ParWithVLSLower;
      A     #VLSLower.InEnableHN;
      O     #VLSLower.StHN;
      );	//[<-4.1]
      =     #VLSUpper.InEnableHN;
      A     #Ma.StOpen;
      AN    #Ma.Par.ParVibroIsMotor;
      AN    #Ma.InDisableVibro;	//[6.2]
      =     #Vibro.InEnableRev;	//FB11.InEnable
      A     #Ma.StOpen;
      A     #Ma.Par.ParVibroIsMotor;
      AN    #Ma.InDisableVibro;	//[6.2]
      =     #Vibro.InEnableFwd;
//--- Sequence Closing ----
      AN    #VLSUpper.InEnableHN;
      =     #VLSUpper.InEnableLN;
      A     #VLSUpper.StLN;
      ON    #Ma.Par.ParWithVLSUpper;
      AN    #tmpOpenReq;
      =     #VLSLower.InEnableLN;
      R     #VLSLower.InEnableHN;
      AN    #Ma.Par.ParWithVLSLower;	//[4.1->]
      A     #VLSLower.InEnableLN;
      O     #VLSLower.StLN;	//[<-4.1]
      AN    #tmpOpenReq;
      =     #AirFlap.InEnableLN;
      R     #AirFlap.InEnableHN;
      =     #AirFlap2.InEnableLN;	//[5.0]
      R     #AirFlap2.InEnableHN;	//[5.0]
// CmdNext
      A     #Ma.CmdNext;	//[6.0]
      ON    #tmpOpenReq;	//[6.0]
      O     #Ma.InManual;	//[6.0]
      S     #AirFlap.CmdNext;
      S     #VLSLower.CmdNext;
      S     #VLSUpper.CmdNext;
      S     #AirFlap2.CmdNext;	//[5.0]
      SET;
      S     #Vibro.CmdNext;
//--- Local mode --
      A     #tmpLocal;
      =     #AirFlap.InLocal;
      =     #VLSLower.InLocal;
      =     #VLSUpper.InLocal;
      =     #AirFlap2.InLocal;	//[5.0]
//--- Fault Reset -------------
      A     #Ma.CmdFaultReset;
      S     #AirFlap.CmdFaultReset;
      S     #VLSLower.CmdFaultReset;
      S     #VLSUpper.CmdFaultReset;
      S     #Vibro.CmdFaultReset;
      S     #AirFlap2.CmdFaultReset;	//[5.0]
NETWORK
TITLE = Call VLS: AirFlap
      AN    #Ma.Par.ParWithAirFlap;
      JC    V2;
      CALL  #AirFlap;
NETWORK
TITLE = Call VLS: AirFlap2 [5.0]
////[5.0] new
      AN    #Ma.Par.ParWithAirFlap2;
      JC    V2;
      CALL  #AirFlap2;
NETWORK
TITLE = Call VLS: VLSLower
V2:   AN    #Ma.Par.ParWithVLSLower;
      JC    V3;
      CALL  #VLSLower;
NETWORK
TITLE = Call VLS: VLSUpper
V3:   AN    #Ma.Par.ParWithVLSUpper;
      JC    V4;
      CALL  #VLSUpper;
NETWORK
TITLE = Call Digital output
V4:   AN    #Ma.Par.ParWithVibro;
      JC    StJ0;
      A     #Ma.Par.ParVibroIsMotor;
      JC    V4M;
      TAR2  #tmpStoreAR2;
      L     P##Vibro;
      L     DW#16#FFFFFF;
      AD;
      +AR2;
      UC    "GCS7_E_DigOutput";	//Call Digital Output FB11
      LAR2  #tmpStoreAR2;
      JU    V4DI;
V4M:  CALL  #Vibro;	//FB12
V4DI: NOP   0;
NETWORK
TITLE = Jump to actual state
StJ0: A     #Ma.StClosed;
      JC    S0;	// ===> State
      A     #Ma.StOpen;
      JC    S2;	// ===> State
      A     #Ma.StOpening;
      JC    S1;	// ===> State
      A     #Ma.StClosing;
      JC    S3;	// ===> State
      A     #Ma.StFault;
      JC    S4;	// ===> State
NETWORK
TITLE = Closed
xxS0: S     #Ma.StClosed;
S0:   R     #Ma.OutPulseClose;	//5.2
      A     #tmpFaultSum;
      R     #Ma.StClosed;
      JC    xxS4;	//--> StFault
// Condition for StOpening
      AN    #AirFlap.StLN;
      A     #Ma.Par.ParWithAirFlap;
      O;
      AN    #AirFlap2.StLN;	//[5.0]
      A     #Ma.Par.ParWithAirFlap2;	//[5.0]
      O;	//[5.0]
      AN    #VLSLower.StLN;
      A     #Ma.Par.ParWithVLSLower;
      O;
      AN    #VLSUpper.StLN;
      A     #Ma.Par.ParWithVLSUpper;
      R     #Ma.StClosed;
      JC    xxS1;	//--> StOpening
      JU    OUT;
NETWORK
TITLE = StOpening
xxS1: S     #Ma.StOpening;
      R     #Ma.OutPulseClose;
S1:   A     #tmpFaultSum;
      R     #Ma.StOpening;
      JC    xxS4;	//--> StFault
// Condition for StClosing
      A     #AirFlap.StLN;
      AN    #AirFlap.OutpLN;
      ON    #Ma.Par.ParWithAirFlap;
      A(;	//[5.0]
      A     #AirFlap2.StLN;	//[5.0]
      AN    #AirFlap2.OutpLN;	//[5.0]
      ON    #Ma.Par.ParWithAirFlap2;	//[5.0]
      );	//[5.0]
      A(;
      A     #VLSLower.StLN;
      AN    #VLSLower.OutpLN;
      ON    #Ma.Par.ParWithVLSLower;
      );
      A(;
      A     #VLSUpper.StLN;
      ON    #Ma.Par.ParWithVLSUpper;
      );
      ON    #tmpOpenReq;
      R     #Ma.StOpening;
      JC    xxS3;	//--> StClosing
// Condition for StOpen
      A     #AirFlap.StHN;
      ON    #Ma.Par.ParWithAirFlap;
      A(;	//[5.0]
      A     #AirFlap2.StHN;	//[5.0]
      ON    #Ma.Par.ParWithAirFlap2;	//[5.0]
      );	//[5.0]
      A(;
      A     #VLSLower.StHN;
      ON    #Ma.Par.ParWithVLSLower;
      );
      A(;
      A     #VLSUpper.StHN;
      ON    #Ma.Par.ParWithVLSUpper;
      );
      R     #Ma.StOpening;
      JC    xxS2;	//--> StOpen
      JU    OUT;
NETWORK
TITLE = StOpen
xxS2: S     #Ma.StOpen;
//Set wait time
      R     #Ma.OutPulseClose;
      L     #Ma.Par.ParWaitOpen;
      T     #Ma.Par.OutTime;
//=== Logic StOpen
S2:   A     #tmpFaultSum;
      R     #Ma.StOpen;
      R     #Ma.OutPulseClose;
      JC    xxS4;	//--> StFault
// Condition for StClosing
      AN    #AirFlap.StHN;
      A     #Ma.Par.ParWithAirFlap;
      O;
      AN    #AirFlap2.StHN;	//[5.0]
      A     #Ma.Par.ParWithAirFlap2;	//[5.0]
      O;	//[5.0]
      AN    #VLSLower.StHN;
      A     #Ma.Par.ParWithVLSLower;
      O;
      AN    #VLSUpper.StHN;
      A     #Ma.Par.ParWithVLSUpper;
      AN    #Ma.Par.ParPulsing;
      O;	//[5.1]
      AN    #VLSUpper.StHN;	//[5.1]
      AN    #tmpOpenReq;	//[5.1]
      A     #Ma.Par.ParWithVLSUpper;	//[5.1]
      R     #Ma.StOpen;
      JC    xxS3;	//--> StClosing
//Pulsing
      A     #Ma.OutPulseClose;
      JC    S2t1;
//===Wait time open
      AN    #VLSUpper.InpHN;
      JC    OUT;
      L     0;
      L     #Ma.Par.OutTime;
      <=I;	//[5.3]   
      JC    S2tx;	//-> Count timer
//Set pulse time close
      S     #Ma.OutPulseClose;
      L     #Ma.Par.ParPulseClosing;
      T     #Ma.Par.OutTime;
      JU    OUT;
//====Pulsing close
S2t1: A     #VLSUpper.InpHN;
      JC    OUT;
      L     0;
      L     #Ma.Par.OutTime;
      <=I;	//[5.3]   
      JC    S2tx;	//-> Count timer
//Set wait time
      R     #Ma.OutPulseClose;
      L     #Ma.Par.ParWaitOpen;
      T     #Ma.Par.OutTime;
      JU    OUT;
//=== Count timer =====
S2tx: AN    "GCS7_Gr_OutTick200ms";	//Gr.OutTick200ms
      JC    OUT;
      L     #Ma.Par.OutTime;
      +     -2;
      T     #Ma.Par.OutTime;
      JU    OUT;
NETWORK
TITLE = StClosing
xxS3: S     #Ma.StClosing;
S3:   A     #tmpFaultSum;
      R     #Ma.StClosing;
      JC    xxS4;	//--> StFault
// Condition for StClosed
      A     #AirFlap.StLN;
      AN    #AirFlap.OutpLN;
      ON    #Ma.Par.ParWithAirFlap;
      A(;	//[5.0]
      A     #AirFlap2.StLN;	//[5.0]
      AN    #AirFlap2.OutpLN;	//[5.0]
      ON    #Ma.Par.ParWithAirFlap2;	//[5.0]
      );	//[5.0]
      A(;
      A     #VLSLower.StLN;
      AN    #VLSLower.OutpLN;
      ON    #Ma.Par.ParWithVLSLower;
      );
      A(;
      A     #VLSUpper.StLN;
      ON    #Ma.Par.ParWithVLSUpper;
      );
      R     #Ma.StClosing;
      JC    xxS0;	//--> StClosed
// Condition for StOpening
      A     #tmpOpenReq;
      R     #Ma.StClosing;
      JC    xxS1;	//--> StOpening
      JU    OUT;
NETWORK
TITLE = Fault
xxS4: S     #Ma.StFault;
S4:   AN    #tmpFaultSum;
      R     #Ma.StFault;
      JC    xxS3;	//--> StClosing
      JU    OUT;
NETWORK
TITLE = Global End
OUT:  CLR;	//---Clear all commands
      =     #Ma.CmdOpen;
      =     #Ma.CmdClose;
      =     #Ma.CmdFaultReset;
      =     #Ma.CmdNext;	//[6.0]
// Disable reading
      A     #VLSUpper.OutpHN;
      AN    #VLSUpper.StHN;
      O;
      A     #VLSUpper.OutpLN;
      AN    #VLSUpper.StLN;
      AN    #VLSUpper.StFault;
      A     #VLSUpper.Par.ParPulseValve;	//[6.1]
      O;	//[6.1]
      A     #VLSUpper.StCtoLN;	//[6.1]
      A     #VLSUpper.Par.ParContValve;	//[6.1]
      =     #Ma.OutDisableRead;
NETWORK
TITLE = State Code
// Same as motor
      A     #Ma.StClosed;
      L     1;	// StCode=Closed
      JC    Code;
      A     #Ma.StOpen;
      L     3;	// StCode=Open
      JC    Code;
      A     #Ma.StOpening;
      L     2;	// StCode=Open
      JC    Code;
      A     #Ma.StClosing;
      L     7;	// StCode=Closing
      JC    Code;
      L     32;	// StCode=Fault
Code: L     #Ma.StCode;	// Old state code
      TAK;
      T     #Ma.StCode;	// Save state code
      <>I;
      L     3;
      CC    "SYS_CBitCtrl";	//Set change bit
END_FUNCTION_BLOCK

